(* IEC 61131-3 sources: verifaps-lib/geteta/examples/RTT_if (part 4) *)

        Pusher_states_t#Reset_interconnect_Slide1_Black:
             a_Pusher$_transit  := FALSE;
             a_Pusher$interconnect3  := FALSE;
             a_Pusher$Timer3$IN  := FALSE;
             a_Pusher$Timer3$PT  := USINT#0;
            IF  a_Pusher$Timer3$IN  THEN
                 a_Pusher$Timer3$Q  := ( a_Pusher$Timer3$ET  = USINT#0);
                IF ( a_Pusher$Timer3$ET  > USINT#0) THEN
                     a_Pusher$Timer3$ET  := ( a_Pusher$Timer3$ET  - USINT#1);
                ELSE
                     a_Pusher$Timer3$ET  := USINT#0;
                END_IF
            ELSE
                 a_Pusher$Timer3$Q  := FALSE;
                 a_Pusher$Timer3$ET  :=  a_Pusher$Timer3$PT ;
            END_IF
             a_Pusher$interconnect_Slide1_Black  := FALSE;
             a_Pusher$Timer_Slide1_Black$IN  := FALSE;
             a_Pusher$Timer_Slide1_Black$PT  := USINT#0;
            IF  a_Pusher$Timer_Slide1_Black$IN  THEN
                 a_Pusher$Timer_Slide1_Black$Q  := ( a_Pusher$Timer_Slide1_Black$ET  = USINT#0);
                IF ( a_Pusher$Timer_Slide1_Black$ET  > USINT#0) THEN
                     a_Pusher$Timer_Slide1_Black$ET  := ( a_Pusher$Timer_Slide1_Black$ET  - USINT#1);
                ELSE
                     a_Pusher$Timer_Slide1_Black$ET  := USINT#0;
                END_IF
            ELSE
                 a_Pusher$Timer_Slide1_Black$Q  := FALSE;
                 a_Pusher$Timer_Slide1_Black$ET  :=  a_Pusher$Timer_Slide1_Black$PT ;
            END_IF
             a_Pusher$Slide1_black  := ( a_Pusher$Slide1_black  - INT#1);
             a_Pusher$Priority_Var_Black  := ( a_Pusher$Priority_Var_Black  - INT#1);
            IF TRUE THEN
                 a_Pusher$_transit  := TRUE;
                 a_Pusher$_state  := Pusher_states_t#Interstep_2;
            END_IF

        Pusher_states_t#Reset_interconnect_Slide1_Metal:
             a_Pusher$_transit  := FALSE;
             a_Pusher$interconnect3  := FALSE;
             a_Pusher$Timer3$IN  := FALSE;
             a_Pusher$Timer3$PT  := USINT#0;
            IF  a_Pusher$Timer3$IN  THEN
                 a_Pusher$Timer3$Q  := ( a_Pusher$Timer3$ET  = USINT#0);
                IF ( a_Pusher$Timer3$ET  > USINT#0) THEN
                     a_Pusher$Timer3$ET  := ( a_Pusher$Timer3$ET  - USINT#1);
                ELSE
                     a_Pusher$Timer3$ET  := USINT#0;
                END_IF
            ELSE
                 a_Pusher$Timer3$Q  := FALSE;
                 a_Pusher$Timer3$ET  :=  a_Pusher$Timer3$PT ;
            END_IF
             a_Pusher$interconnect_Slide1_Metal  := FALSE;
             a_Pusher$Timer_Slide1_Metal$IN  := FALSE;
             a_Pusher$Timer_Slide1_Metal$PT  := USINT#0;
            IF  a_Pusher$Timer_Slide1_Metal$IN  THEN
                 a_Pusher$Timer_Slide1_Metal$Q  := ( a_Pusher$Timer_Slide1_Metal$ET  = USINT#0);
                IF ( a_Pusher$Timer_Slide1_Metal$ET  > USINT#0) THEN
                     a_Pusher$Timer_Slide1_Metal$ET  := ( a_Pusher$Timer_Slide1_Metal$ET  - USINT#1);
                ELSE
                     a_Pusher$Timer_Slide1_Metal$ET  := USINT#0;
                END_IF
            ELSE
                 a_Pusher$Timer_Slide1_Metal$Q  := FALSE;
                 a_Pusher$Timer_Slide1_Metal$ET  :=  a_Pusher$Timer_Slide1_Metal$PT ;
            END_IF
             a_Pusher$Slide1_metal  := ( a_Pusher$Slide1_metal  - INT#1);
             a_Pusher$Priority_Var_Metal  := ( a_Pusher$Priority_Var_Metal  - INT#1);
            IF TRUE THEN
                 a_Pusher$_transit  := TRUE;
                 a_Pusher$_state  := Pusher_states_t#Interstep_2;
            END_IF

        Pusher_states_t#Reset_interconnect_Slide1_White:
             a_Pusher$_transit  := FALSE;
             a_Pusher$interconnect3  := FALSE;
             a_Pusher$Timer3$IN  := FALSE;
             a_Pusher$Timer3$PT  := USINT#0;
            IF  a_Pusher$Timer3$IN  THEN
                 a_Pusher$Timer3$Q  := ( a_Pusher$Timer3$ET  = USINT#0);
                IF ( a_Pusher$Timer3$ET  > USINT#0) THEN
                     a_Pusher$Timer3$ET  := ( a_Pusher$Timer3$ET  - USINT#1);
                ELSE
                     a_Pusher$Timer3$ET  := USINT#0;
                END_IF
            ELSE
                 a_Pusher$Timer3$Q  := FALSE;
                 a_Pusher$Timer3$ET  :=  a_Pusher$Timer3$PT ;
            END_IF
             a_Pusher$interconnect_Slide1_White  := FALSE;
             a_Pusher$Timer_Slide1_White$IN  := FALSE;
             a_Pusher$Timer_Slide1_White$PT  := USINT#0;
            IF  a_Pusher$Timer_Slide1_White$IN  THEN
                 a_Pusher$Timer_Slide1_White$Q  := ( a_Pusher$Timer_Slide1_White$ET  = USINT#0);
                IF ( a_Pusher$Timer_Slide1_White$ET  > USINT#0) THEN
                     a_Pusher$Timer_Slide1_White$ET  := ( a_Pusher$Timer_Slide1_White$ET  - USINT#1);
                ELSE
                     a_Pusher$Timer_Slide1_White$ET  := USINT#0;
                END_IF
            ELSE
                 a_Pusher$Timer_Slide1_White$Q  := FALSE;
                 a_Pusher$Timer_Slide1_White$ET  :=  a_Pusher$Timer_Slide1_White$PT ;
            END_IF
             a_Pusher$Slide1_white  := ( a_Pusher$Slide1_white  - INT#1);
             a_Pusher$Priority_Var_White  := ( a_Pusher$Priority_Var_White  - INT#1);
            IF TRUE THEN
                 a_Pusher$_transit  := TRUE;
                 a_Pusher$_state  := Pusher_states_t#Interstep_2;
            END_IF

        Pusher_states_t#Reset_interconnect_Slide2_Black:
             a_Pusher$_transit  := FALSE;
             a_Pusher$interconnect3  := FALSE;
             a_Pusher$Timer3$IN  := FALSE;
             a_Pusher$Timer3$PT  := USINT#0;
            IF  a_Pusher$Timer3$IN  THEN
                 a_Pusher$Timer3$Q  := ( a_Pusher$Timer3$ET  = USINT#0);
                IF ( a_Pusher$Timer3$ET  > USINT#0) THEN
                     a_Pusher$Timer3$ET  := ( a_Pusher$Timer3$ET  - USINT#1);
                ELSE
                     a_Pusher$Timer3$ET  := USINT#0;
                END_IF
            ELSE
                 a_Pusher$Timer3$Q  := FALSE;
                 a_Pusher$Timer3$ET  :=  a_Pusher$Timer3$PT ;
            END_IF
             a_Pusher$interconnect_Slide2_Black  := FALSE;
             a_Pusher$Timer_Slide2_Black$IN  := FALSE;
             a_Pusher$Timer_Slide2_Black$PT  := USINT#0;
            IF  a_Pusher$Timer_Slide2_Black$IN  THEN
                 a_Pusher$Timer_Slide2_Black$Q  := ( a_Pusher$Timer_Slide2_Black$ET  = USINT#0);
                IF ( a_Pusher$Timer_Slide2_Black$ET  > USINT#0) THEN
                     a_Pusher$Timer_Slide2_Black$ET  := ( a_Pusher$Timer_Slide2_Black$ET  - USINT#1);
                ELSE
                     a_Pusher$Timer_Slide2_Black$ET  := USINT#0;
                END_IF
            ELSE
                 a_Pusher$Timer_Slide2_Black$Q  := FALSE;
                 a_Pusher$Timer_Slide2_Black$ET  :=  a_Pusher$Timer_Slide2_Black$PT ;
            END_IF
             a_Pusher$Slide2_black  := ( a_Pusher$Slide2_black  - INT#1);
             a_Pusher$Priority_Var_Black  := ( a_Pusher$Priority_Var_Black  - INT#1);
            IF TRUE THEN
                 a_Pusher$_transit  := TRUE;
                 a_Pusher$_state  := Pusher_states_t#Interstep_2;
            END_IF

        Pusher_states_t#Reset_interconnect_Slide2_Metal:
             a_Pusher$_transit  := FALSE;
             a_Pusher$interconnect3  := FALSE;
             a_Pusher$Timer3$IN  := FALSE;
             a_Pusher$Timer3$PT  := USINT#0;
            IF  a_Pusher$Timer3$IN  THEN
                 a_Pusher$Timer3$Q  := ( a_Pusher$Timer3$ET  = USINT#0);
                IF ( a_Pusher$Timer3$ET  > USINT#0) THEN
                     a_Pusher$Timer3$ET  := ( a_Pusher$Timer3$ET  - USINT#1);
                ELSE
                     a_Pusher$Timer3$ET  := USINT#0;
                END_IF
            ELSE
                 a_Pusher$Timer3$Q  := FALSE;
                 a_Pusher$Timer3$ET  :=  a_Pusher$Timer3$PT ;
            END_IF
             a_Pusher$interconnect_Slide2_Metal  := FALSE;
             a_Pusher$Timer_Slide2_Metal$IN  := FALSE;
             a_Pusher$Timer_Slide2_Metal$PT  := USINT#0;
            IF  a_Pusher$Timer_Slide2_Metal$IN  THEN
                 a_Pusher$Timer_Slide2_Metal$Q  := ( a_Pusher$Timer_Slide2_Metal$ET  = USINT#0);
                IF ( a_Pusher$Timer_Slide2_Metal$ET  > USINT#0) THEN
                     a_Pusher$Timer_Slide2_Metal$ET  := ( a_Pusher$Timer_Slide2_Metal$ET  - USINT#1);
                ELSE
                     a_Pusher$Timer_Slide2_Metal$ET  := USINT#0;
                END_IF
            ELSE
                 a_Pusher$Timer_Slide2_Metal$Q  := FALSE;
                 a_Pusher$Timer_Slide2_Metal$ET  :=  a_Pusher$Timer_Slide2_Metal$PT ;
            END_IF
             a_Pusher$Slide2_metal  := ( a_Pusher$Slide2_metal  - INT#1);
             a_Pusher$Priority_Var_Metal  := ( a_Pusher$Priority_Var_Metal  - INT#1);
            IF TRUE THEN
                 a_Pusher$_transit  := TRUE;
                 a_Pusher$_state  := Pusher_states_t#Interstep_2;
            END_IF

        Pusher_states_t#Reset_interconnect_Slide2_White:
             a_Pusher$_transit  := FALSE;
             a_Pusher$interconnect3  := FALSE;
             a_Pusher$Timer3$IN  := FALSE;
             a_Pusher$Timer3$PT  := USINT#0;
            IF  a_Pusher$Timer3$IN  THEN
                 a_Pusher$Timer3$Q  := ( a_Pusher$Timer3$ET  = USINT#0);
                IF ( a_Pusher$Timer3$ET  > USINT#0) THEN
                     a_Pusher$Timer3$ET  := ( a_Pusher$Timer3$ET  - USINT#1);
                ELSE
                     a_Pusher$Timer3$ET  := USINT#0;
                END_IF
            ELSE
                 a_Pusher$Timer3$Q  := FALSE;
                 a_Pusher$Timer3$ET  :=  a_Pusher$Timer3$PT ;
            END_IF
             a_Pusher$interconnect_Slide2_White  := FALSE;
             a_Pusher$Timer_Slide2_White$IN  := FALSE;
             a_Pusher$Timer_Slide2_White$PT  := USINT#0;
            IF  a_Pusher$Timer_Slide2_White$IN  THEN
                 a_Pusher$Timer_Slide2_White$Q  := ( a_Pusher$Timer_Slide2_White$ET  = USINT#0);
                IF ( a_Pusher$Timer_Slide2_White$ET  > USINT#0) THEN
                     a_Pusher$Timer_Slide2_White$ET  := ( a_Pusher$Timer_Slide2_White$ET  - USINT#1);
                ELSE
                     a_Pusher$Timer_Slide2_White$ET  := USINT#0;
                END_IF
            ELSE
                 a_Pusher$Timer_Slide2_White$Q  := FALSE;
                 a_Pusher$Timer_Slide2_White$ET  :=  a_Pusher$Timer_Slide2_White$PT ;
            END_IF
             a_Pusher$Slide2_white  := ( a_Pusher$Slide2_white  - INT#1);
             a_Pusher$Priority_Var_White  := ( a_Pusher$Priority_Var_White  - INT#1);
            IF TRUE THEN
                 a_Pusher$_transit  := TRUE;
                 a_Pusher$_state  := Pusher_states_t#Interstep_2;
            END_IF

        Pusher_states_t#Reset_interconnect_Slide3_Metal:
             a_Pusher$_transit  := FALSE;
             a_Pusher$interconnect3  := FALSE;
             a_Pusher$Timer3$IN  := FALSE;
             a_Pusher$Timer3$PT  := USINT#0;
            IF  a_Pusher$Timer3$IN  THEN
                 a_Pusher$Timer3$Q  := ( a_Pusher$Timer3$ET  = USINT#0);
                IF ( a_Pusher$Timer3$ET  > USINT#0) THEN
                     a_Pusher$Timer3$ET  := ( a_Pusher$Timer3$ET  - USINT#1);
                ELSE
                     a_Pusher$Timer3$ET  := USINT#0;
                END_IF
            ELSE
                 a_Pusher$Timer3$Q  := FALSE;
                 a_Pusher$Timer3$ET  :=  a_Pusher$Timer3$PT ;
            END_IF
             a_Pusher$Slide3_metal  := ( a_Pusher$Slide3_metal  - INT#1);
             a_Pusher$Priority_Var_Metal  := ( a_Pusher$Priority_Var_Metal  - INT#1);
            IF TRUE THEN
                 a_Pusher$_transit  := TRUE;
                 a_Pusher$_state  := Pusher_states_t#Interstep_2;
            END_IF

        Pusher_states_t#Reset_interconnect_Slide3_White:
             a_Pusher$_transit  := FALSE;
             a_Pusher$interconnect3  := FALSE;
             a_Pusher$Timer3$IN  := FALSE;
             a_Pusher$Timer3$PT  := USINT#0;
            IF  a_Pusher$Timer3$IN  THEN
                 a_Pusher$Timer3$Q  := ( a_Pusher$Timer3$ET  = USINT#0);
                IF ( a_Pusher$Timer3$ET  > USINT#0) THEN
                     a_Pusher$Timer3$ET  := ( a_Pusher$Timer3$ET  - USINT#1);
                ELSE
                     a_Pusher$Timer3$ET  := USINT#0;
                END_IF
            ELSE
                 a_Pusher$Timer3$Q  := FALSE;
                 a_Pusher$Timer3$ET  :=  a_Pusher$Timer3$PT ;
            END_IF
             a_Pusher$Slide3_white  := ( a_Pusher$Slide3_white  - INT#1);
             a_Pusher$Priority_Var_White  := ( a_Pusher$Priority_Var_White  - INT#1);
            IF TRUE THEN
                 a_Pusher$_transit  := TRUE;
                 a_Pusher$_state  := Pusher_states_t#Interstep_2;
            END_IF

        Pusher_states_t#Second_Slide_Timer_Black:
             a_Pusher$_transit  := FALSE;
            IF ( a_Pusher$SorterLightnesssensorCraneInterfaceInverse  = TRUE) THEN
                 a_Pusher$Timer_Slide2_Black$IN  :=  a_Pusher$SorterLightnesssensorCraneInterfaceInverse ;
                 a_Pusher$Timer_Slide2_Black$PT  :=  a_Pusher$Duration_Slide2_Black ;
                IF  a_Pusher$Timer_Slide2_Black$IN  THEN
                     a_Pusher$Timer_Slide2_Black$Q  := ( a_Pusher$Timer_Slide2_Black$ET  = USINT#0);
                    IF ( a_Pusher$Timer_Slide2_Black$ET  > USINT#0) THEN
                         a_Pusher$Timer_Slide2_Black$ET  := ( a_Pusher$Timer_Slide2_Black$ET  - USINT#1);
                    ELSE
                         a_Pusher$Timer_Slide2_Black$ET  := USINT#0;
                    END_IF
                ELSE
                     a_Pusher$Timer_Slide2_Black$Q  := FALSE;
                     a_Pusher$Timer_Slide2_Black$ET  :=  a_Pusher$Timer_Slide2_Black$PT ;
                END_IF
                 a_Pusher$interconnect_Slide2_Black  :=  a_Pusher$Timer_Slide2_Black$Q ;
            END_IF
            IF  a_Pusher$interconnect_Slide2_Black  THEN
                 a_Pusher$_transit  := TRUE;
                 a_Pusher$_state  := Pusher_states_t#PusherY2_Move_Out_Black;
            END_IF

        Pusher_states_t#Second_Slide_Timer_Metal:
             a_Pusher$_transit  := FALSE;
             a_Pusher$Timer_Slide2_Metal$IN  := TRUE;
             a_Pusher$Timer_Slide2_Metal$PT  :=  a_Pusher$Duration_Slide2_Metal ;
            IF  a_Pusher$Timer_Slide2_Metal$IN  THEN
                 a_Pusher$Timer_Slide2_Metal$Q  := ( a_Pusher$Timer_Slide2_Metal$ET  = USINT#0);
                IF ( a_Pusher$Timer_Slide2_Metal$ET  > USINT#0) THEN
                     a_Pusher$Timer_Slide2_Metal$ET  := ( a_Pusher$Timer_Slide2_Metal$ET  - USINT#1);
                ELSE
                     a_Pusher$Timer_Slide2_Metal$ET  := USINT#0;
                END_IF
            ELSE
                 a_Pusher$Timer_Slide2_Metal$Q  := FALSE;
                 a_Pusher$Timer_Slide2_Metal$ET  :=  a_Pusher$Timer_Slide2_Metal$PT ;
            END_IF
             a_Pusher$interconnect_Slide2_Metal  :=  a_Pusher$Timer_Slide2_Metal$Q ;
            IF  a_Pusher$interconnect_Slide2_Metal  THEN
                 a_Pusher$_transit  := TRUE;
                 a_Pusher$_state  := Pusher_states_t#PusherY2_Move_Out_Metal;
            END_IF

        Pusher_states_t#Second_Slide_Timer_White:
             a_Pusher$_transit  := FALSE;
             a_Pusher$Timer_Slide2_White$IN  := TRUE;
             a_Pusher$Timer_Slide2_White$PT  :=  a_Pusher$Duration_Slide2_White ;
            IF  a_Pusher$Timer_Slide2_White$IN  THEN
                 a_Pusher$Timer_Slide2_White$Q  := ( a_Pusher$Timer_Slide2_White$ET  = USINT#0);
                IF ( a_Pusher$Timer_Slide2_White$ET  > USINT#0) THEN
                     a_Pusher$Timer_Slide2_White$ET  := ( a_Pusher$Timer_Slide2_White$ET  - USINT#1);
                ELSE
                     a_Pusher$Timer_Slide2_White$ET  := USINT#0;
                END_IF
            ELSE
                 a_Pusher$Timer_Slide2_White$Q  := FALSE;
                 a_Pusher$Timer_Slide2_White$ET  :=  a_Pusher$Timer_Slide2_White$PT ;
            END_IF
             a_Pusher$interconnect_Slide2_White  :=  a_Pusher$Timer_Slide2_White$Q ;
            IF  a_Pusher$interconnect_Slide2_White  THEN
                 a_Pusher$_transit  := TRUE;
                 a_Pusher$_state  := Pusher_states_t#PusherY2_Move_Out_White;
            END_IF

        Pusher_states_t#Second_Slide_black_workpieces:
             a_Pusher$_transit  := FALSE;
            IF TRUE THEN
                 a_Pusher$_transit  := TRUE;
                 a_Pusher$_state  := Pusher_states_t#Second_Slide_Timer_Black;
            END_IF

        Pusher_states_t#Second_Slide_metal_workpieces:
             a_Pusher$_transit  := FALSE;
            IF ( a_Pusher$SorterLightnessSensorPusher2  AND  a_Pusher$SorterCapacitiveSensorPusher2 ) THEN
                 a_Pusher$_transit  := TRUE;
                 a_Pusher$_state  := Pusher_states_t#Second_Test_For_Metal;
            END_IF

        Pusher_states_t#Second_Slide_white_workpieces:
             a_Pusher$_transit  := FALSE;
            IF ( a_Pusher$SorterLightnessSensorPusher2  AND NOT  a_Pusher$SorterCapacitiveSensorPusher2 ) THEN
                 a_Pusher$_transit  := TRUE;
                 a_Pusher$_state  := Pusher_states_t#Second_Test_For_White;
            END_IF

        Pusher_states_t#Second_Test_For_Metal:
             a_Pusher$_transit  := FALSE;
            IF TRUE THEN
                 a_Pusher$_transit  := TRUE;
                 a_Pusher$_state  := Pusher_states_t#Second_Slide_Timer_Metal;
            END_IF

        Pusher_states_t#Second_Test_For_White:
             a_Pusher$_transit  := FALSE;
            IF TRUE THEN
                 a_Pusher$_transit  := TRUE;
                 a_Pusher$_state  := Pusher_states_t#Second_Slide_Timer_White;
            END_IF

        Pusher_states_t#Third_Slide_black_workpieces:
             a_Pusher$_transit  := FALSE;
            IF (NOT  a_Pusher$SorterLightnessSensorPusher2  AND NOT  a_Pusher$SorterCapacitiveSensorPusher2 ) THEN
                 a_Pusher$_transit  := TRUE;
                 a_Pusher$_state  := Pusher_states_t#Wait_Black;
            END_IF

        Pusher_states_t#Third_Slide_metal_workpieces:
             a_Pusher$_transit  := FALSE;
            IF ( a_Pusher$SorterLightnessSensorPusher2  AND  a_Pusher$SorterCapacitiveSensorPusher2 ) THEN
                 a_Pusher$_transit  := TRUE;
                 a_Pusher$_state  := Pusher_states_t#Wait_Metal;
            END_IF

        Pusher_states_t#Third_Slide_white_workpieces:
             a_Pusher$_transit  := FALSE;
            IF ( a_Pusher$SorterLightnessSensorPusher2  AND NOT  a_Pusher$SorterCapacitiveSensorPusher2 ) THEN
                 a_Pusher$_transit  := TRUE;
                 a_Pusher$_state  := Pusher_states_t#Wait_White;
            END_IF

        Pusher_states_t#Wait_Black:
             a_Pusher$_transit  := FALSE;
            IF ((NOT  a_Pusher$SorterLightnessSensorPusher2  AND NOT  a_Pusher$SorterCapacitiveSensorPusher2 ) = TRUE) THEN
                 a_Pusher$Timer2$IN  := (NOT  a_Pusher$SorterLightnessSensorPusher2  AND NOT  a_Pusher$SorterCapacitiveSensorPusher2 );
                 a_Pusher$Timer2$PT  :=  a_Pusher$Duration2 ;
                IF  a_Pusher$Timer2$IN  THEN
                     a_Pusher$Timer2$Q  := ( a_Pusher$Timer2$ET  = USINT#0);
                    IF ( a_Pusher$Timer2$ET  > USINT#0) THEN
                         a_Pusher$Timer2$ET  := ( a_Pusher$Timer2$ET  - USINT#1);
                    ELSE
                         a_Pusher$Timer2$ET  := USINT#0;
                    END_IF
                ELSE
                     a_Pusher$Timer2$Q  := FALSE;
                     a_Pusher$Timer2$ET  :=  a_Pusher$Timer2$PT ;
                END_IF
                 a_Pusher$interconnect2  :=  a_Pusher$Timer2$Q ;
            END_IF
            IF  a_Pusher$interconnect2  THEN
                 a_Pusher$_transit  := TRUE;
                 a_Pusher$_state  := Pusher_states_t#Reset_interconnect3;
            END_IF

        Pusher_states_t#Wait_Metal:
             a_Pusher$_transit  := FALSE;
             a_Pusher$Timer3$IN  := TRUE;
             a_Pusher$Timer3$PT  :=  a_Pusher$Duration3 ;
            IF  a_Pusher$Timer3$IN  THEN
                 a_Pusher$Timer3$Q  := ( a_Pusher$Timer3$ET  = USINT#0);
                IF ( a_Pusher$Timer3$ET  > USINT#0) THEN
                     a_Pusher$Timer3$ET  := ( a_Pusher$Timer3$ET  - USINT#1);
                ELSE
                     a_Pusher$Timer3$ET  := USINT#0;
                END_IF
            ELSE
                 a_Pusher$Timer3$Q  := FALSE;
                 a_Pusher$Timer3$ET  :=  a_Pusher$Timer3$PT ;
            END_IF
             a_Pusher$interconnect3  :=  a_Pusher$Timer3$Q ;
            IF  a_Pusher$interconnect3  THEN
                 a_Pusher$_transit  := TRUE;
                 a_Pusher$_state  := Pusher_states_t#Reset_interconnect_Slide3_Metal;
            END_IF

        Pusher_states_t#Wait_White:
             a_Pusher$_transit  := FALSE;
             a_Pusher$Timer3$IN  := TRUE;
             a_Pusher$Timer3$PT  :=  a_Pusher$Duration3 ;
            IF  a_Pusher$Timer3$IN  THEN
                 a_Pusher$Timer3$Q  := ( a_Pusher$Timer3$ET  = USINT#0);
                IF ( a_Pusher$Timer3$ET  > USINT#0) THEN
                     a_Pusher$Timer3$ET  := ( a_Pusher$Timer3$ET  - USINT#1);
                ELSE
                     a_Pusher$Timer3$ET  := USINT#0;
                END_IF
            ELSE
                 a_Pusher$Timer3$Q  := FALSE;
                 a_Pusher$Timer3$ET  :=  a_Pusher$Timer3$PT ;
            END_IF
             a_Pusher$interconnect3  :=  a_Pusher$Timer3$Q ;
            IF  a_Pusher$interconnect3  THEN
                 a_Pusher$_transit  := TRUE;
                 a_Pusher$_state  := Pusher_states_t#Reset_interconnect_Slide3_White;
            END_IF

        Pusher_states_t#Wait_Y1_Black:
             a_Pusher$_transit  := FALSE;
            IF ( a_Pusher$PusherY1  = TRUE) THEN
                 a_Pusher$Timer3$IN  :=  a_Pusher$PusherY1 ;
                 a_Pusher$Timer3$PT  :=  a_Pusher$Duration3 ;
                IF  a_Pusher$Timer3$IN  THEN
                     a_Pusher$Timer3$Q  := ( a_Pusher$Timer3$ET  = USINT#0);
                    IF ( a_Pusher$Timer3$ET  > USINT#0) THEN
                         a_Pusher$Timer3$ET  := ( a_Pusher$Timer3$ET  - USINT#1);
                    ELSE
                         a_Pusher$Timer3$ET  := USINT#0;
                    END_IF
                ELSE
                     a_Pusher$Timer3$Q  := FALSE;
                     a_Pusher$Timer3$ET  :=  a_Pusher$Timer3$PT ;
                END_IF
                 a_Pusher$interconnect3  :=  a_Pusher$Timer3$Q ;
            END_IF
            IF  a_Pusher$interconnect3  THEN
                 a_Pusher$_transit  := TRUE;
                 a_Pusher$_state  := Pusher_states_t#PusherY1_Move_In_Black;
            END_IF

        Pusher_states_t#Wait_Y1_Metal:
             a_Pusher$_transit  := FALSE;
            IF ( a_Pusher$PusherY1  = TRUE) THEN
                 a_Pusher$Timer3$IN  :=  a_Pusher$PusherY1 ;
                 a_Pusher$Timer3$PT  :=  a_Pusher$Duration3 ;
                IF  a_Pusher$Timer3$IN  THEN
                     a_Pusher$Timer3$Q  := ( a_Pusher$Timer3$ET  = USINT#0);
                    IF ( a_Pusher$Timer3$ET  > USINT#0) THEN
                         a_Pusher$Timer3$ET  := ( a_Pusher$Timer3$ET  - USINT#1);
                    ELSE
                         a_Pusher$Timer3$ET  := USINT#0;
                    END_IF
                ELSE
                     a_Pusher$Timer3$Q  := FALSE;
                     a_Pusher$Timer3$ET  :=  a_Pusher$Timer3$PT ;
                END_IF
                 a_Pusher$interconnect3  :=  a_Pusher$Timer3$Q ;
            END_IF
            IF  a_Pusher$interconnect3  THEN
                 a_Pusher$_transit  := TRUE;
                 a_Pusher$_state  := Pusher_states_t#PusherY1_Move_In_Metal;
            END_IF

        Pusher_states_t#Wait_Y1_White:
             a_Pusher$_transit  := FALSE;
            IF ( a_Pusher$PusherY1  = TRUE) THEN
                 a_Pusher$Timer3$IN  :=  a_Pusher$PusherY1 ;
                 a_Pusher$Timer3$PT  :=  a_Pusher$Duration3 ;
                IF  a_Pusher$Timer3$IN  THEN
                     a_Pusher$Timer3$Q  := ( a_Pusher$Timer3$ET  = USINT#0);
                    IF ( a_Pusher$Timer3$ET  > USINT#0) THEN
                         a_Pusher$Timer3$ET  := ( a_Pusher$Timer3$ET  - USINT#1);
                    ELSE
                         a_Pusher$Timer3$ET  := USINT#0;
                    END_IF
                ELSE
                     a_Pusher$Timer3$Q  := FALSE;
                     a_Pusher$Timer3$ET  :=  a_Pusher$Timer3$PT ;
                END_IF
                 a_Pusher$interconnect3  :=  a_Pusher$Timer3$Q ;
            END_IF
            IF  a_Pusher$interconnect3  THEN
                 a_Pusher$_transit  := TRUE;
                 a_Pusher$_state  := Pusher_states_t#PusherY1_Move_In_White;
            END_IF

        Pusher_states_t#Wait_Y2_Black:
             a_Pusher$_transit  := FALSE;
            IF ( a_Pusher$PusherY2  = TRUE) THEN
                 a_Pusher$Timer3$IN  :=  a_Pusher$PusherY2 ;
                 a_Pusher$Timer3$PT  :=  a_Pusher$Duration3 ;
                IF  a_Pusher$Timer3$IN  THEN
                     a_Pusher$Timer3$Q  := ( a_Pusher$Timer3$ET  = USINT#0);
                    IF ( a_Pusher$Timer3$ET  > USINT#0) THEN
                         a_Pusher$Timer3$ET  := ( a_Pusher$Timer3$ET  - USINT#1);
                    ELSE
                         a_Pusher$Timer3$ET  := USINT#0;
                    END_IF
                ELSE
                     a_Pusher$Timer3$Q  := FALSE;
                     a_Pusher$Timer3$ET  :=  a_Pusher$Timer3$PT ;
                END_IF
                 a_Pusher$interconnect3  :=  a_Pusher$Timer3$Q ;
            END_IF
            IF  a_Pusher$interconnect3  THEN
                 a_Pusher$_transit  := TRUE;
                 a_Pusher$_state  := Pusher_states_t#PusherY2_Move_In_Black;
            END_IF

        Pusher_states_t#Wait_Y2_Metal:
             a_Pusher$_transit  := FALSE;
            IF ( a_Pusher$PusherY2  = TRUE) THEN
                 a_Pusher$Timer3$IN  :=  a_Pusher$PusherY2 ;
                 a_Pusher$Timer3$PT  :=  a_Pusher$Duration3 ;
                IF  a_Pusher$Timer3$IN  THEN
                     a_Pusher$Timer3$Q  := ( a_Pusher$Timer3$ET  = USINT#0);
                    IF ( a_Pusher$Timer3$ET  > USINT#0) THEN
                         a_Pusher$Timer3$ET  := ( a_Pusher$Timer3$ET  - USINT#1);
                    ELSE
                         a_Pusher$Timer3$ET  := USINT#0;
                    END_IF
                ELSE
                     a_Pusher$Timer3$Q  := FALSE;
                     a_Pusher$Timer3$ET  :=  a_Pusher$Timer3$PT ;
                END_IF
                 a_Pusher$interconnect3  :=  a_Pusher$Timer3$Q ;
            END_IF
            IF  a_Pusher$interconnect3  THEN
                 a_Pusher$_transit  := TRUE;
                 a_Pusher$_state  := Pusher_states_t#PusherY2_Move_In_Metal;
            END_IF

        Pusher_states_t#Wait_Y2_White:
             a_Pusher$_transit  := FALSE;
            IF ( a_Pusher$PusherY2  = TRUE) THEN
                 a_Pusher$Timer3$IN  :=  a_Pusher$PusherY2 ;
                 a_Pusher$Timer3$PT  :=  a_Pusher$Duration3 ;
                IF  a_Pusher$Timer3$IN  THEN
                     a_Pusher$Timer3$Q  := ( a_Pusher$Timer3$ET  = USINT#0);
                    IF ( a_Pusher$Timer3$ET  > USINT#0) THEN
                         a_Pusher$Timer3$ET  := ( a_Pusher$Timer3$ET  - USINT#1);
                    ELSE
                         a_Pusher$Timer3$ET  := USINT#0;
                    END_IF
                ELSE
                     a_Pusher$Timer3$Q  := FALSE;
                     a_Pusher$Timer3$ET  :=  a_Pusher$Timer3$PT ;
                END_IF
                 a_Pusher$interconnect3  :=  a_Pusher$Timer3$Q ;
            END_IF
            IF  a_Pusher$interconnect3  THEN
                 a_Pusher$_transit  := TRUE;
                 a_Pusher$_state  := Pusher_states_t#PusherY2_Move_In_White;
            END_IF

            END_CASE
    IF (( a_Actuator_SorterGreenLampConveyor  AND  a_Actuator_MagazinGreenLamp ) AND  a_Actuator_StampGreenLamp ) THEN
        IF ((( a_Stamp$StartCommandStamp  AND  a_Crane$StartCommandCrane ) AND  a_Conveyor$StartCommandConveyor ) AND  a_Mag$StartCommandMagazin ) THEN
             a_Crane$StartVar  := TRUE;
             a_Conveyor$StartVar  := TRUE;
             a_Mag$StartVar  := TRUE;
             a_Pusher$StartVar  := TRUE;
             a_Stamp$StartVar  := TRUE;
             a_DIAGNOSIS_ACTIVE  := TRUE;
        END_IF
    END_IF
     a_Crane$SFCReset  := FALSE;
     a_Conveyor$SFCReset  := FALSE;
     a_Mag$SFCReset  := FALSE;
     a_Pusher$SFCReset  := FALSE;
     a_Stamp$SFCReset  := FALSE;

     a_Crane$AnalogCranePressure  :=  a_PARAMETER_CRANE_PRESSURE_METALLIC ;

ELSEIF ((NOT  a_Sensor_SorterEmergencyStop  OR NOT  a_Sensor_StampEmergencyStop ) OR NOT  a_Sensor_MagazinEmergencyStop ) THEN
     a_Actuator_MagazinSlider  := FALSE;
     a_Actuator_CraneLower  := FALSE;
     a_Actuator_MagazinVacuumOn  := FALSE;
     a_Actuator_MagazinVacuumOff  := TRUE;
     a_Actuator_MagazinGreenLamp  := FALSE;
     a_Actuator_CraneTurnCounterclockwise  := FALSE;
     a_Actuator_CraneTurnClockwise  := FALSE;
     a_Actuator_SorterConveyorTowardsStacker  := FALSE;
     a_Actuator_SorterConveyorTowardsCrane  := FALSE;
     a_Actuator_SorterGreenLampConveyor  := FALSE;
     a_Actuator_PusherY1  := FALSE;
     a_Actuator_PusherY2  := FALSE;
     a_Actuator_StampSliderMovedOut  := TRUE;
     a_Actuator_StampSliderMovedIn  := FALSE;
     a_Actuator_StampGreenLamp  := FALSE;
     a_Actuator_StampPusher  := FALSE;
     a_Actuator_AnalogCranePressure  := INT#0;
     a_Crane$SFCReset  := TRUE;
     a_Conveyor$SFCReset  := TRUE;
     a_Mag$SFCReset  := TRUE;
     a_Pusher$SFCReset  := TRUE;
     a_Stamp$SFCReset  := TRUE;
     a_Crane$StartVar  := FALSE;
     a_Conveyor$StartVar  := FALSE;
     a_Mag$StartVar  := FALSE;
     a_Pusher$StartVar  := FALSE;
     a_Stamp$StartVar  := FALSE;
END_IF

//--------------------------------------------------------------------------------

 b_Mag$SliderNotMovedOut  :=  b_Sensor_SliderNotMovedOut ;
 b_Mag$SliderMovedOut  :=  b_Sensor_SliderMovedOut ;
 b_Mag$CraneOnMagazin  :=  b_Sensor_CraneOnMagazin ;
 b_Mag$CraneDown  :=  b_Sensor_CraneDown ;
 b_Mag$CraneUp  :=  b_Sensor_CraneUp ;
 b_Mag$CraneOnConveyor  :=  b_Sensor_CraneOnConveyor ;
 b_Mag$WorkpieceReady  :=  b_Sensor_WorkpieceReady ;
 b_Mag$AnalogCranePosition  :=  b_Sensor_AnalogCranePosition ;
 b_Mag$StartButtonMagazin  :=  b_Sensor_StartButtonMagazin ;
 b_Actuator_MagazinSlider  :=  b_Mag$MagazinSlider ;
 b_Actuator_MagazinGreenLamp  :=  b_Mag$MagazinGreenLamp ;
 b_Crane$CraneUp  :=  b_Sensor_CraneUp ;
 b_Crane$CraneDown  :=  b_Sensor_CraneDown ;
 b_Crane$CraneSucked  :=  b_Sensor_CraneSucked ;
 b_Crane$MagazinCapacitiveSensor  :=  b_Sensor_MagazinCapacitiveSensor ;
 b_Crane$SliderMovedOut  :=  b_Sensor_SliderMovedOut ;
 b_Crane$WorkpieceReady  :=  b_Sensor_WorkpieceReady ;
 b_Crane$MagazinOpticalSensor  :=  b_Sensor_MagazinOpticalSensor ;
 b_Crane$StampSliderFilled  :=  b_Sensor_StampSliderFilled ;
 b_Crane$StampSliderSensorMovedOut  :=  b_Sensor_StampSliderSensorMovedOut ;
 b_Crane$StampLowered  :=  b_Sensor_StampLowered ;
 b_Crane$AnalogCranePosition  :=  b_Sensor_AnalogCranePosition ;
 b_Crane$StartButtonMagazin  :=  b_Sensor_StartButtonMagazin ;

//Diagnosis
// old:  b_Actuator_AnalogCranePressure
// new:  b_Crane$AnalogCranePressure ;
 b_Actuator_CraneTurnCounterclockwise  :=  b_Crane$CraneTurnCounterclockwise ;
 b_Actuator_CraneTurnClockwise  :=  b_Crane$CraneTurnClockwise ;

IF  b_DIAGNOSIS_ACTIVE  THEN
        IF  b_Sensor_CraneSucked  AND ( b_Crane$AnalogCranePressure  <= 0 OR  b_Crane$AnalogCranePressure  > 10000) THEN
                 b_Actuator_CraneTurnCounterclockwise  := FALSE;
                 b_Actuator_CraneTurnClockwise  := FALSE;
        END_IF
END_IF

//End of Diagnosis

 b_Actuator_CraneLower  :=  b_Crane$CraneLower ;
 b_Actuator_MagazinVacuumOff  :=  b_Crane$MagazinVacuumOff ;
 b_Actuator_MagazinVacuumOn  :=  b_Crane$MagazinVacuumOn ;
 b_Actuator_AnalogCranePressure  :=  b_Crane$AnalogCranePressure ;
 b_Stamp$StampSliderSensorMovedOut  :=  b_Sensor_StampSliderSensorMovedOut ;
 b_Stamp$StampSliderSensorMovedIn  :=  b_Sensor_StampSliderSensorMovedIn ;
 b_Stamp$StampSliderFilled  :=  b_Sensor_StampSliderFilled ;
 b_Stamp$StampUp  :=  b_Sensor_StampUp ;
 b_Stamp$StampLowered  :=  b_Sensor_StampLowered ;
 b_Stamp$CraneDown  :=  b_Sensor_CraneDown ;
 b_Stamp$CraneUp  :=  b_Sensor_CraneUp ;
 b_Stamp$CraneSucked  :=  b_Sensor_CraneSucked ;
 b_Stamp$CranePositionStamp  :=  b_Sensor_CranePositionStamp ;
 b_Stamp$CraneOnConveyor  :=  b_Sensor_CraneOnConveyor ;
 b_Stamp$AnalogCranePosition  :=  b_Sensor_AnalogCranePosition ;
 b_Stamp$StampStartButton  :=  b_Sensor_StampStartButton ;
 b_Actuator_StampSliderMovedOut  :=  b_Stamp$StampSliderMovedOut ;
 b_Actuator_StampSliderMovedIn  :=  b_Stamp$StampSliderMovedIn ;
 b_Actuator_StampWhiteLamp  :=  b_Stamp$StampWhiteLamp ;
 b_Actuator_StampPusher  :=  b_Stamp$StampPusher ;
 b_Actuator_StampGreenLamp  :=  b_Stamp$StampGreenLamp ;
 b_Conveyor$SorterStartButton  :=  b_Sensor_SorterStartButton ;
 b_Conveyor$SorterSwitchManuellAutomatic  :=  b_Sensor_SorterSwitchManuellAutomatic ;
 b_Conveyor$SorterLightbarrierCraneInterface  :=  b_Sensor_SorterLightbarrierCraneInterface ;
 b_Actuator_SorterConveyorTowardsStacker  :=  b_Conveyor$SorterConveyorTowardsStacker ;
 b_Actuator_SorterConveyorTowardsCrane  :=  b_Conveyor$SorterConveyorTowardsCrane ;
 b_Actuator_SorterGreenLampConveyor  :=  b_Conveyor$SorterGreenLampConveyor ;
 b_Actuator_SorterWhiteLampConveyor  :=  b_Conveyor$SorterWhiteLampConveyor ;
 b_Pusher$SorterLightnesssensorCraneInterfaceInverse  :=  b_Sensor_SorterLightnesssensorCraneInterfaceInverse ;
 b_Pusher$SorterLightbarrierCraneInterface  :=  b_Sensor_SorterLightbarrierCraneInterface ;
 b_Pusher$SorterCapacitiveSensorPusher1  :=  b_Sensor_SorterCapacitiveSensorPusher1 ;
 b_Pusher$SorterLightnessSensorPusher1  :=  b_Sensor_SorterLightnessSensorPusher1 ;
 b_Pusher$SorterCapacitiveSensorPusher2  :=  b_Sensor_SorterCapacitiveSensorPusher2 ;
 b_Pusher$SorterLightnessSensorPusher2  :=  b_Sensor_SorterLightnessSensorPusher2 ;
 b_Pusher$SorterLightnessSensorPusher3  :=  b_Sensor_SorterLightnessSensorPusher3 ;
 b_Pusher$SorterPusher1MovedOut  :=  b_Sensor_SorterPusher1MovedOut ;
 b_Pusher$SorterPusher1MovedIn  :=  b_Sensor_SorterPusher1MovedIn ;
 b_Pusher$SorterPusher2MovedOut  :=  b_Sensor_SorterPusher2MovedOut ;
 b_Pusher$SorterPusher2MovedIn  :=  b_Sensor_SorterPusher2MovedIn ;
 b_Pusher$SorterStartButton  :=  b_Sensor_SorterStartButton ;
 b_Actuator_PusherY1  :=  b_Pusher$PusherY1 ;
 b_Actuator_PusherY2  :=  b_Pusher$PusherY2 ;

IF (( b_Sensor_SorterEmergencyStop  AND  b_Sensor_StampEmergencyStop ) AND  b_Sensor_MagazinEmergencyStop ) THEN
    CASE  b_Mag$_state  OF
        Magazin_states_t#Green_Lamp:
             b_Mag$_transit  := FALSE;
             b_Mag$MagazinGreenLamp  := TRUE;
             b_Mag$interconnectMagazinStartCommand  := FALSE;
            IF TRUE THEN
                 b_Mag$_transit  := TRUE;
                 b_Mag$_state  := Magazin_states_t#Magazin_Init;
            END_IF

        Magazin_states_t#Init:
             b_Mag$_transit  := FALSE;
            IF TRUE THEN
                 b_Mag$_transit  := TRUE;
                 b_Mag$_state  := Magazin_states_t#Start_Magazin;
            END_IF

        Magazin_states_t#Interstep:
             b_Mag$_transit  := FALSE;
             b_Mag$StartCommandMagazin  := TRUE;
            IF  b_Mag$StartVar  THEN
                 b_Mag$_transit  := TRUE;
                 b_Mag$_state  := Magazin_states_t#convey;
            END_IF

        Magazin_states_t#Magazin_Init:
             b_Mag$_transit  := FALSE;
             b_Mag$MagazinSlider  := TRUE;
            IF TRUE THEN
                 b_Mag$_transit  := TRUE;
                 b_Mag$_state  := Magazin_states_t#Magazin_Init_2;
            END_IF

        Magazin_states_t#Magazin_Init_2:
             b_Mag$_transit  := FALSE;
             b_Mag$MagazinSlider  := FALSE;
            IF TRUE THEN
                 b_Mag$_transit  := TRUE;
                 b_Mag$_state  := Magazin_states_t#Interstep;
            END_IF

        Magazin_states_t#Slider_Move_Back:
             b_Mag$_transit  := FALSE;
            IF (( b_Mag$SliderMovedOut  = TRUE) AND ( b_Mag$SliderNotMovedOut  = FALSE)) THEN
                 b_Mag$MagazinSlider  := FALSE;
            END_IF
            IF  b_Mag$CraneUp  THEN
                 b_Mag$_transit  := TRUE;
                 b_Mag$_state  := Magazin_states_t#Step1;
            END_IF

        Magazin_states_t#Start_Magazin:
             b_Mag$_transit  := FALSE;
             b_Mag$MagazinSlider  := FALSE;
             b_Mag$MagazinGreenLamp  := FALSE;
             b_Mag$StartVar  := FALSE;
             b_Mag$StartCommandMagazin  := FALSE;
            IF ( b_Mag$StartButtonMagazin  = TRUE) THEN
                 b_Mag$interconnectMagazinStartCommand  := TRUE;
            END_IF
            IF  b_Mag$interconnectMagazinStartCommand  THEN
                 b_Mag$_transit  := TRUE;
                 b_Mag$_state  := Magazin_states_t#Green_Lamp;
            END_IF

        Magazin_states_t#Step0:
             b_Mag$_transit  := FALSE;
            IF  b_Mag$CraneDown  THEN
                 b_Mag$_transit  := TRUE;
                 b_Mag$_state  := Magazin_states_t#Slider_Move_Back;
            END_IF

        Magazin_states_t#Step1:
             b_Mag$_transit  := FALSE;
            IF (( b_Mag$AnalogCranePosition  > INT#16160) AND ( b_Mag$AnalogCranePosition  < INT#16260)) THEN
                 b_Mag$_transit  := TRUE;
                 b_Mag$_state  := Magazin_states_t#Interstep;
            END_IF

        Magazin_states_t#convey:
             b_Mag$_transit  := FALSE;
            IF  b_Mag$SliderNotMovedOut  THEN
                 b_Mag$MagazinSlider  := TRUE;
            END_IF
            IF (( b_Mag$AnalogCranePosition  > INT#24290) AND ( b_Mag$AnalogCranePosition  < INT#24390)) THEN
                 b_Mag$_transit  := TRUE;
                 b_Mag$_state  := Magazin_states_t#Step0;
            END_IF

            END_CASE
    CASE  b_Crane$_state  OF
        Crane_states_t#Crane_Go_Up:
             b_Crane$_transit  := FALSE;
             b_Crane$CraneLower  := FALSE;
            IF  b_Crane$CraneUp  THEN
                 b_Crane$_transit  := TRUE;
                 b_Crane$_state  := Crane_states_t#Step3;
            END_IF

        Crane_states_t#Crane_Go_Up_White:
             b_Crane$_transit  := FALSE;
             b_Crane$CraneLower  := FALSE;
            IF  b_Crane$CraneUp  THEN
                 b_Crane$_transit  := TRUE;
                 b_Crane$_state  := Crane_states_t#Step3;
            END_IF

        Crane_states_t#Crane_Init:
             b_Crane$_transit  := FALSE;
             b_Crane$CraneLower  := TRUE;
             b_Crane$interconnectCraneStartCommand  := FALSE;
             b_Crane$AnalogCranePressure  :=  b_PARAMETER_CRANE_PRESSURE_METALLIC ;
            IF  b_Crane$CraneDown  THEN
                 b_Crane$_transit  := TRUE;
                 b_Crane$_state  := Crane_states_t#Crane_Init_2;
            END_IF

        Crane_states_t#Crane_Init_2:
             b_Crane$_transit  := FALSE;
             b_Crane$CraneLower  := FALSE;
            IF  b_Crane$CraneUp  THEN
                 b_Crane$_transit  := TRUE;
                 b_Crane$_state  := Crane_states_t#Interstep;
            END_IF

        Crane_states_t#Crane_Lift_At_Stamp:
             b_Crane$_transit  := FALSE;
             b_Crane$CraneLower  := FALSE;
            IF  b_Crane$CraneUp  THEN
                 b_Crane$_transit  := TRUE;
                 b_Crane$_state  := Crane_states_t#Crane_Turn_Left_From_Stamp;
            END_IF

        Crane_states_t#Crane_Lift_At_Stamp2:
             b_Crane$_transit  := FALSE;
             b_Crane$CraneLower  := FALSE;
             b_Crane$AnalogCranePressure  := INT#0;
            IF  b_Crane$CraneUp  THEN
                 b_Crane$_transit  := TRUE;
                 b_Crane$_state  := Crane_states_t#Crane_Turn_Right_From_Stamp;
            END_IF

        Crane_states_t#Crane_Lift_Conveyor:
             b_Crane$_transit  := FALSE;
             b_Crane$CraneLower  := FALSE;
            IF TRUE THEN
                 b_Crane$_transit  := TRUE;
                 b_Crane$_state  := Crane_states_t#Interstep;
            END_IF

        Crane_states_t#Crane_Lift_Conveyor2:
             b_Crane$_transit  := FALSE;
             b_Crane$CraneLower  := FALSE;
            IF TRUE THEN
                 b_Crane$_transit  := TRUE;
                 b_Crane$_state  := Crane_states_t#Interstep;
            END_IF

        Crane_states_t#Crane_Lift_Conveyor_Black:
             b_Crane$_transit  := FALSE;
             b_Crane$CraneLower  := FALSE;
            IF  b_Crane$CraneUp  THEN
                 b_Crane$_transit  := TRUE;
                 b_Crane$_state  := Crane_states_t#Crane_Turn_Left_Back_To_Stamp;
            END_IF

        Crane_states_t#Crane_Lift_Magazin:
             b_Crane$_transit  := FALSE;
             b_Crane$CraneLower  := FALSE;
            IF  b_Crane$CraneUp  THEN
                 b_Crane$_transit  := TRUE;
                 b_Crane$_state  := Crane_states_t#Crane_Turn_Left_NOT_Metallic;
            END_IF

        Crane_states_t#Crane_Lift_Magazin_Metallic:
             b_Crane$_transit  := FALSE;
             b_Crane$CraneLower  := FALSE;
            IF  b_Crane$CraneUp  THEN
                 b_Crane$_transit  := TRUE;
                 b_Crane$_state  := Crane_states_t#Crane_Turn_Left_Metallic;
            END_IF

        Crane_states_t#Crane_Lift_Magazin_White:
             b_Crane$_transit  := FALSE;
             b_Crane$CraneLower  := FALSE;
            IF  b_Crane$CraneUp  THEN
                 b_Crane$_transit  := TRUE;
                 b_Crane$_state  := Crane_states_t#Crane_Turn_Left_White;
            END_IF

        Crane_states_t#Crane_Lift_NOT_Metallic_Black:
             b_Crane$_transit  := FALSE;
             b_Crane$CraneLower  := FALSE;
            IF  b_Crane$CraneUp  THEN
                 b_Crane$_transit  := TRUE;
                 b_Crane$_state  := Crane_states_t#Crane_Turn_Left_NOT_Metallic_Black;
            END_IF

        Crane_states_t#Crane_Lower:
             b_Crane$_transit  := FALSE;
             b_Crane$MagazinVacuumOn  := TRUE;
             b_Crane$MagazinVacuumOff  := FALSE;
             b_Crane$CraneLower  := TRUE;
             b_Crane$AnalogCranePressure  := INT#0;
            IF  b_Crane$CraneSucked  THEN
                 b_Crane$_transit  := TRUE;
                 b_Crane$_state  := Crane_states_t#Step0;
            END_IF

        Crane_states_t#Crane_On_Conveyor:
             b_Crane$_transit  := FALSE;
             b_Crane$CraneTurnCounterclockwise  := FALSE;
             b_Crane$CraneTurnClockwise  := FALSE;
             b_Crane$CraneLower  := TRUE;
            IF  b_Crane$CraneDown  THEN
                 b_Crane$_transit  := TRUE;
                 b_Crane$_state  := Crane_states_t#release;
            END_IF

        Crane_states_t#Crane_On_Conveyor_Metallic:
             b_Crane$_transit  := FALSE;
             b_Crane$CraneTurnCounterclockwise  := FALSE;
             b_Crane$CraneTurnClockwise  := FALSE;
             b_Crane$CraneLower  := TRUE;
            IF  b_Crane$CraneDown  THEN
                 b_Crane$_transit  := TRUE;
                 b_Crane$_state  := Crane_states_t#release;
            END_IF

        Crane_states_t#Crane_On_Conveyor_Metallic2:
             b_Crane$_transit  := FALSE;
             b_Crane$CraneTurnCounterclockwise  := FALSE;
             b_Crane$CraneTurnClockwise  := FALSE;
             b_Crane$CraneLower  := TRUE;
            IF  b_Crane$CraneDown  THEN
                 b_Crane$_transit  := TRUE;
                 b_Crane$_state  := Crane_states_t#release2;
            END_IF

        Crane_states_t#Crane_On_Conveyor_Not_Metallica_Black:
             b_Crane$_transit  := FALSE;
             b_Crane$CraneTurnCounterclockwise  := FALSE;
             b_Crane$CraneTurnClockwise  := FALSE;
             b_Crane$CraneLower  := TRUE;
            IF  b_Crane$CraneDown  THEN
                 b_Crane$_transit  := TRUE;
                 b_Crane$_state  := Crane_states_t#release_Black;
            END_IF

        Crane_states_t#Crane_On_Stamp_Metallic:
             b_Crane$_transit  := FALSE;
             b_Crane$CraneTurnCounterclockwise  := FALSE;
             b_Crane$CraneTurnClockwise  := FALSE;
             b_Crane$CraneLower  := TRUE;
            IF  b_Crane$CraneDown  THEN
                 b_Crane$_transit  := TRUE;
                 b_Crane$_state  := Crane_states_t#release_Workpiece;
            END_IF

        Crane_states_t#Crane_On_Stamp_Metallic2:
             b_Crane$_transit  := FALSE;
             b_Crane$CraneTurnCounterclockwise  := FALSE;
             b_Crane$CraneTurnClockwise  := FALSE;
            IF  b_Crane$StampLowered  THEN
                 b_Crane$_transit  := TRUE;
                 b_Crane$_state  := Crane_states_t#Interstep_4;
            END_IF

        Crane_states_t#Crane_On_Stamp_Metallic2_Lower:
             b_Crane$_transit  := FALSE;
             b_Crane$CraneLower  := TRUE;
            IF  b_Crane$CraneDown  THEN
                 b_Crane$_transit  := TRUE;
                 b_Crane$_state  := Crane_states_t#Suck_At_Stamp2;
            END_IF

        Crane_states_t#Crane_On_Stamp_Stop_Black:
             b_Crane$_transit  := FALSE;
             b_Crane$CraneTurnClockwise  := FALSE;
             b_Crane$CraneTurnCounterclockwise  := FALSE;
            IF TRUE THEN
                 b_Crane$_transit  := TRUE;
                 b_Crane$_state  := Crane_states_t#Reset_interconnect;
            END_IF

        Crane_states_t#Crane_On_Stamp_White:
             b_Crane$_transit  := FALSE;
             b_Crane$CraneTurnCounterclockwise  := FALSE;
             b_Crane$CraneTurnClockwise  := FALSE;
             b_Crane$CraneLower  := TRUE;
            IF  b_Crane$CraneDown  THEN
                 b_Crane$_transit  := TRUE;
                 b_Crane$_state  := Crane_states_t#release_Workpiece_White;
            END_IF

        Crane_states_t#Crane_Turn_Left_Back_To_Stamp:
             b_Crane$_transit  := FALSE;
             b_Crane$CraneTurnCounterclockwise  := TRUE;
             b_Crane$CraneTurnClockwise  := FALSE;
            IF (( b_Crane$AnalogCranePosition  > INT#8160) AND ( b_Crane$AnalogCranePosition  < INT#8260)) THEN
                 b_Crane$_transit  := TRUE;
                 b_Crane$_state  := Crane_states_t#Crane_On_Stamp_Stop_Black;
            END_IF

        Crane_states_t#Crane_Turn_Left_From_Stamp:
             b_Crane$_transit  := FALSE;
             b_Crane$CraneTurnClockwise  := TRUE;
             b_Crane$CraneTurnCounterclockwise  := FALSE;
            IF (( b_Crane$AnalogCranePosition  > INT#16060) AND ( b_Crane$AnalogCranePosition  < INT#16160)) THEN
                 b_Crane$_transit  := TRUE;
                 b_Crane$_state  := Crane_states_t#Crane_On_Conveyor_Metallic;
            END_IF

        Crane_states_t#Crane_Turn_Left_Metallic:
             b_Crane$_transit  := FALSE;
             b_Crane$CraneTurnCounterclockwise  := TRUE;
             b_Crane$CraneTurnClockwise  := FALSE;
            IF (( b_Crane$AnalogCranePosition  > INT#8160) AND ( b_Crane$AnalogCranePosition  < INT#8260)) THEN
                 b_Crane$_transit  := TRUE;
                 b_Crane$_state  := Crane_states_t#Crane_On_Stamp_Metallic;
            END_IF

        Crane_states_t#Crane_Turn_Left_Metallic2:
             b_Crane$_transit  := FALSE;
             b_Crane$CraneTurnCounterclockwise  := TRUE;
             b_Crane$CraneTurnClockwise  := FALSE;
            IF (( b_Crane$AnalogCranePosition  > INT#8160) AND ( b_Crane$AnalogCranePosition  < INT#8260)) THEN
                 b_Crane$_transit  := TRUE;
                 b_Crane$_state  := Crane_states_t#Crane_On_Stamp_Metallic2;
            END_IF

        Crane_states_t#Crane_Turn_Left_NOT_Metallic:
             b_Crane$_transit  := FALSE;
             b_Crane$CraneTurnCounterclockwise  := TRUE;
             b_Crane$CraneTurnClockwise  := FALSE;
            IF (( b_Crane$AnalogCranePosition  > INT#16160) AND ( b_Crane$AnalogCranePosition  < INT#16260)) THEN
                 b_Crane$_transit  := TRUE;
                 b_Crane$_state  := Crane_states_t#Crane_On_Conveyor;
            END_IF

        Crane_states_t#Crane_Turn_Left_NOT_Metallic_Black:
             b_Crane$_transit  := FALSE;
             b_Crane$CraneTurnCounterclockwise  := TRUE;
             b_Crane$CraneTurnClockwise  := FALSE;
            IF (( b_Crane$AnalogCranePosition  > INT#16160) AND ( b_Crane$AnalogCranePosition  < INT#16260)) THEN
                 b_Crane$_transit  := TRUE;
                 b_Crane$_state  := Crane_states_t#Crane_On_Conveyor_Not_Metallica_Black;
            END_IF

        Crane_states_t#Crane_Turn_Left_White:
             b_Crane$_transit  := FALSE;
             b_Crane$CraneTurnCounterclockwise  := TRUE;
             b_Crane$CraneTurnClockwise  := FALSE;
            IF (( b_Crane$AnalogCranePosition  > INT#8160) AND ( b_Crane$AnalogCranePosition  < INT#8260)) THEN
                 b_Crane$_transit  := TRUE;
                 b_Crane$_state  := Crane_states_t#Crane_On_Stamp_White;
            END_IF

        Crane_states_t#Crane_Turn_Right_From_Stamp:
             b_Crane$_transit  := FALSE;
             b_Crane$CraneTurnClockwise  := TRUE;
             b_Crane$CraneTurnCounterclockwise  := FALSE;
            IF (( b_Crane$AnalogCranePosition  > INT#16160) AND ( b_Crane$AnalogCranePosition  < INT#16260)) THEN
                 b_Crane$_transit  := TRUE;
                 b_Crane$_state  := Crane_states_t#Crane_On_Conveyor_Metallic2;
            END_IF

        Crane_states_t#Init:
             b_Crane$_transit  := FALSE;
            IF TRUE THEN
                 b_Crane$_transit  := TRUE;
                 b_Crane$_state  := Crane_states_t#Start_Crane;
            END_IF

        Crane_states_t#Interstep:
             b_Crane$_transit  := FALSE;
             b_Crane$StartCommandCrane  := TRUE;
            IF  b_Crane$StartVar  THEN
                 b_Crane$_transit  := TRUE;
                 b_Crane$_state  := Crane_states_t#Interstep_2;
            END_IF

        Crane_states_t#Interstep_2:
             b_Crane$_transit  := FALSE;
            IF  b_Crane$SliderMovedOut  THEN
                 b_Crane$_transit  := TRUE;
                 b_Crane$_state  := Crane_states_t#TimeDelay;
            END_IF

        Crane_states_t#Interstep_3:
             b_Crane$_transit  := FALSE;
            IF NOT  b_Crane$WorkpieceReady  THEN
                 b_Crane$_transit  := TRUE;
                 b_Crane$_state  := Crane_states_t#No_Workpiece_ready;
            ELSEIF  b_Crane$WorkpieceReady  THEN
                 b_Crane$_transit  := TRUE;
                 b_Crane$_state  := Crane_states_t#Turn_Right;
            END_IF

        Crane_states_t#Interstep_4:
             b_Crane$_transit  := FALSE;
            IF  b_Crane$StampSliderSensorMovedOut  THEN
                 b_Crane$_transit  := TRUE;
                 b_Crane$_state  := Crane_states_t#Crane_On_Stamp_Metallic2_Lower;
            END_IF

        Crane_states_t#Lower_Crane:
             b_Crane$_transit  := FALSE;
             b_Crane$CraneLower  := TRUE;
            IF  b_Crane$CraneDown  THEN
                 b_Crane$_transit  := TRUE;
                 b_Crane$_state  := Crane_states_t#Suck_At_Stamp;
            END_IF

        Crane_states_t#Magazin_Stop:
             b_Crane$_transit  := FALSE;
             b_Crane$CraneTurnClockwise  := FALSE;
             b_Crane$CraneTurnCounterclockwise  := FALSE;
            IF TRUE THEN
                 b_Crane$_transit  := TRUE;
                 b_Crane$_state  := Crane_states_t#Crane_Lower;
            END_IF

        Crane_states_t#Magazin_Stop_Black:
             b_Crane$_transit  := FALSE;
             b_Crane$CraneTurnClockwise  := FALSE;
             b_Crane$CraneTurnCounterclockwise  := FALSE;
             b_Crane$MagazinVacuumOn  := TRUE;
             b_Crane$MagazinVacuumOff  := FALSE;
             b_Crane$CraneLower  := TRUE;
            IF  b_Crane$CraneSucked  THEN
                 b_Crane$_transit  := TRUE;
                 b_Crane$_state  := Crane_states_t#Crane_Lift_NOT_Metallic_Black;
            END_IF

        Crane_states_t#Magazin_Stop_Final:
             b_Crane$_transit  := FALSE;
             b_Crane$CraneTurnClockwise  := FALSE;
             b_Crane$CraneTurnCounterclockwise  := FALSE;
            IF TRUE THEN
                 b_Crane$_transit  := TRUE;
                 b_Crane$_state  := Crane_states_t#Start_Crane;
            END_IF

        Crane_states_t#No_Workpiece_ready:
             b_Crane$_transit  := FALSE;
             b_Crane$MagazinVacuumOn  := FALSE;
             b_Crane$MagazinVacuumOff  := FALSE;
             b_Crane$CraneLower  := FALSE;
            IF  b_Crane$StampSliderFilled  THEN
                 b_Crane$_transit  := TRUE;
                 b_Crane$_state  := Crane_states_t#Crane_Turn_Left_Metallic2;
            ELSEIF NOT  b_Crane$StampSliderFilled  THEN
                 b_Crane$_transit  := TRUE;
                 b_Crane$_state  := Crane_states_t#Turn_Right_Final;
            END_IF

        Crane_states_t#Reset_interconnect:
             b_Crane$_transit  := FALSE;
             b_Crane$interconnect  := FALSE;
             b_Crane$Timer1$IN  := FALSE;
             b_Crane$Timer1$PT  := USINT#0;
            IF  b_Crane$Timer1$IN  THEN
                 b_Crane$Timer1$Q  := ( b_Crane$Timer1$ET  = USINT#0);
                IF ( b_Crane$Timer1$ET  > USINT#0) THEN
                     b_Crane$Timer1$ET  := ( b_Crane$Timer1$ET  - USINT#1);
                ELSE
                     b_Crane$Timer1$ET  := USINT#0;
                END_IF
            ELSE
                 b_Crane$Timer1$Q  := FALSE;
                 b_Crane$Timer1$ET  :=  b_Crane$Timer1$PT ;
            END_IF
            IF  b_Crane$SliderMovedOut  THEN
                 b_Crane$_transit  := TRUE;
                 b_Crane$_state  := Crane_states_t#Lower_Crane;
            END_IF

        Crane_states_t#Stamp_Pressure_Profile_Set_Metallic:
             b_Crane$_transit  := FALSE;
             b_Crane$AnalogCranePressure  :=  b_PARAMETER_CRANE_PRESSURE_METALLIC ;
            IF TRUE THEN
                 b_Crane$_transit  := TRUE;
                 b_Crane$_state  := Crane_states_t#Crane_Lift_Magazin_Metallic;
            END_IF

        Crane_states_t#Stamp_Pressure_Profile_Set_White:
             b_Crane$_transit  := FALSE;
             b_Crane$AnalogCranePressure  :=  b_PARAMETER_CRANE_PRESSURE_WHITE ;
            IF TRUE THEN
                 b_Crane$_transit  := TRUE;
                 b_Crane$_state  := Crane_states_t#Crane_Lift_Magazin_White;
            END_IF

        Crane_states_t#Start_Crane:
             b_Crane$_transit  := FALSE;
             b_Crane$CraneLower  := FALSE;
             b_Crane$MagazinVacuumOff  := FALSE;
             b_Crane$MagazinVacuumOn  := FALSE;
             b_Crane$CraneTurnCounterclockwise  := FALSE;
             b_Crane$CraneTurnClockwise  := FALSE;
             b_Crane$AnalogCranePressure  := INT#0;
             b_Crane$StartVar  := FALSE;
             b_Crane$StartCommandCrane  := FALSE;
            IF ( b_Crane$StartButtonMagazin  = TRUE) THEN
                 b_Crane$interconnectCraneStartCommand  := TRUE;
            END_IF
            IF  b_Crane$interconnectCraneStartCommand  THEN
                 b_Crane$_transit  := TRUE;
                 b_Crane$_state  := Crane_states_t#Crane_Init;
            END_IF

        Crane_states_t#Step0:
             b_Crane$_transit  := FALSE;
            IF ( b_Crane$MagazinCapacitiveSensor  AND  b_Crane$MagazinOpticalSensor ) THEN
                 b_Crane$_transit  := TRUE;
                 b_Crane$_state  := Crane_states_t#Stamp_Pressure_Profile_Set_Metallic;
            ELSEIF (NOT  b_Crane$MagazinCapacitiveSensor  AND  b_Crane$MagazinOpticalSensor ) THEN
                 b_Crane$_transit  := TRUE;
                 b_Crane$_state  := Crane_states_t#Stamp_Pressure_Profile_Set_White;
            ELSEIF (NOT  b_Crane$MagazinCapacitiveSensor  AND NOT  b_Crane$MagazinOpticalSensor ) THEN
                 b_Crane$_transit  := TRUE;
                 b_Crane$_state  := Crane_states_t#Crane_Lift_Magazin;
            END_IF

        Crane_states_t#Step2:
             b_Crane$_transit  := FALSE;
            IF ( b_Crane$MagazinCapacitiveSensor  OR  b_Crane$MagazinOpticalSensor ) THEN
                 b_Crane$_transit  := TRUE;
                 b_Crane$_state  := Crane_states_t#pause;
            ELSEIF (NOT  b_Crane$MagazinCapacitiveSensor  AND NOT  b_Crane$MagazinOpticalSensor ) THEN
                 b_Crane$_transit  := TRUE;
                 b_Crane$_state  := Crane_states_t#Turn_Right_Black;
            END_IF

        Crane_states_t#Step3:
             b_Crane$_transit  := FALSE;
            IF NOT  b_Crane$WorkpieceReady  THEN
                 b_Crane$_transit  := TRUE;
                 b_Crane$_state  := Crane_states_t#Step4;
            ELSEIF  b_Crane$WorkpieceReady  THEN
                 b_Crane$_transit  := TRUE;
                 b_Crane$_state  := Crane_states_t#Step2;
            END_IF

        Crane_states_t#Step4:
             b_Crane$_transit  := FALSE;
            IF TRUE THEN
                 b_Crane$_transit  := TRUE;
                 b_Crane$_state  := Crane_states_t#Interstep;
            END_IF

        Crane_states_t#Suck_At_Stamp:
             b_Crane$_transit  := FALSE;
             b_Crane$MagazinVacuumOn  := TRUE;
             b_Crane$MagazinVacuumOff  := FALSE;
            IF  b_Crane$CraneSucked  THEN
                 b_Crane$_transit  := TRUE;
                 b_Crane$_state  := Crane_states_t#Crane_Lift_At_Stamp;
            END_IF

        Crane_states_t#Suck_At_Stamp2:
             b_Crane$_transit  := FALSE;
             b_Crane$MagazinVacuumOn  := TRUE;
             b_Crane$MagazinVacuumOff  := FALSE;
            IF  b_Crane$CraneSucked  THEN
                 b_Crane$_transit  := TRUE;
                 b_Crane$_state  := Crane_states_t#Crane_Lift_At_Stamp2;
            END_IF

        Crane_states_t#TimeDelay:
             b_Crane$_transit  := FALSE;
             b_Crane$TimeDelay_Timer$IN  := TRUE;
             b_Crane$TimeDelay_Timer$PT  :=  b_Crane$TimeDelay_Timer_Duration ;
            IF  b_Crane$TimeDelay_Timer$IN  THEN
                 b_Crane$TimeDelay_Timer$Q  := ( b_Crane$TimeDelay_Timer$ET  = USINT#0);
                IF ( b_Crane$TimeDelay_Timer$ET  > USINT#0) THEN
                     b_Crane$TimeDelay_Timer$ET  := ( b_Crane$TimeDelay_Timer$ET  - USINT#1);
                ELSE
                     b_Crane$TimeDelay_Timer$ET  := USINT#0;
                END_IF
            ELSE
                 b_Crane$TimeDelay_Timer$Q  := FALSE;
                 b_Crane$TimeDelay_Timer$ET  :=  b_Crane$TimeDelay_Timer$PT ;
            END_IF
             b_Crane$TimeDelay_Timer_interconnect  :=  b_Crane$TimeDelay_Timer$Q ;
            IF  b_Crane$TimeDelay_Timer_interconnect  THEN
                 b_Crane$_transit  := TRUE;
                 b_Crane$_state  := Crane_states_t#Interstep_3;
            END_IF

        Crane_states_t#Turn_Right:
             b_Crane$_transit  := FALSE;
             b_Crane$CraneTurnClockwise  := TRUE;
             b_Crane$CraneTurnCounterclockwise  := FALSE;
            IF (( b_Crane$AnalogCranePosition  > INT#24290) AND ( b_Crane$AnalogCranePosition  < INT#24390)) THEN
                 b_Crane$_transit  := TRUE;
                 b_Crane$_state  := Crane_states_t#Magazin_Stop;
            END_IF

        Crane_states_t#Turn_Right_Black:
             b_Crane$_transit  := FALSE;
             b_Crane$CraneTurnClockwise  := TRUE;
             b_Crane$CraneTurnCounterclockwise  := FALSE;
            IF (( b_Crane$AnalogCranePosition  > INT#24290) AND ( b_Crane$AnalogCranePosition  < INT#24390)) THEN
                 b_Crane$_transit  := TRUE;
                 b_Crane$_state  := Crane_states_t#Magazin_Stop_Black;
            END_IF

        Crane_states_t#Turn_Right_Final:
             b_Crane$_transit  := FALSE;
             b_Crane$CraneTurnClockwise  := TRUE;
             b_Crane$CraneTurnCounterclockwise  := FALSE;
             b_Crane$AnalogCranePressure  := INT#0;
            IF (( b_Crane$AnalogCranePosition  > INT#24290) AND ( b_Crane$AnalogCranePosition  < INT#24390)) THEN
                 b_Crane$_transit  := TRUE;
                 b_Crane$_state  := Crane_states_t#Magazin_Stop_Final;
            END_IF

        Crane_states_t#pause:
             b_Crane$_transit  := FALSE;
             b_Crane$Timer1$IN  :=  b_Crane$CraneUp ;
             b_Crane$Timer1$PT  :=  b_Crane$Duration1 ;
            IF  b_Crane$Timer1$IN  THEN
                 b_Crane$Timer1$Q  := ( b_Crane$Timer1$ET  = USINT#0);
                IF ( b_Crane$Timer1$ET  > USINT#0) THEN
                     b_Crane$Timer1$ET  := ( b_Crane$Timer1$ET  - USINT#1);
                ELSE
                     b_Crane$Timer1$ET  := USINT#0;
                END_IF
            ELSE
                 b_Crane$Timer1$Q  := FALSE;
                 b_Crane$Timer1$ET  :=  b_Crane$Timer1$PT ;
            END_IF
             b_Crane$interconnect  :=  b_Crane$Timer1$Q ;
            IF  b_Crane$interconnect  THEN
                 b_Crane$_transit  := TRUE;
                 b_Crane$_state  := Crane_states_t#Reset_interconnect;
            END_IF

        Crane_states_t#release:
             b_Crane$_transit  := FALSE;
             b_Crane$MagazinVacuumOff  := TRUE;
             b_Crane$MagazinVacuumOn  := FALSE;
            IF TRUE THEN
                 b_Crane$_transit  := TRUE;
                 b_Crane$_state  := Crane_states_t#Crane_Lift_Conveyor;
            END_IF

        Crane_states_t#release2:
             b_Crane$_transit  := FALSE;
             b_Crane$MagazinVacuumOff  := TRUE;
             b_Crane$MagazinVacuumOn  := FALSE;
            IF TRUE THEN
                 b_Crane$_transit  := TRUE;
                 b_Crane$_state  := Crane_states_t#Crane_Lift_Conveyor2;
            END_IF

        Crane_states_t#release_Black:
             b_Crane$_transit  := FALSE;
             b_Crane$MagazinVacuumOn  := FALSE;
             b_Crane$MagazinVacuumOff  := TRUE;
            IF TRUE THEN
                 b_Crane$_transit  := TRUE;
                 b_Crane$_state  := Crane_states_t#Crane_Lift_Conveyor_Black;
            END_IF

        Crane_states_t#release_Workpiece:
             b_Crane$_transit  := FALSE;
             b_Crane$MagazinVacuumOff  := TRUE;
             b_Crane$MagazinVacuumOn  := FALSE;
            IF TRUE THEN
                 b_Crane$_transit  := TRUE;
                 b_Crane$_state  := Crane_states_t#Crane_Go_Up;
            END_IF

        Crane_states_t#release_Workpiece_White:
             b_Crane$_transit  := FALSE;
             b_Crane$MagazinVacuumOff  := TRUE;
             b_Crane$MagazinVacuumOn  := FALSE;
            IF TRUE THEN
                 b_Crane$_transit  := TRUE;
                 b_Crane$_state  := Crane_states_t#Crane_Go_Up_White;
            END_IF

            END_CASE
    CASE  b_Stamp$_state  OF
        Stamp_states_t#Green_Lamp:
             b_Stamp$_transit  := FALSE;
             b_Stamp$StampGreenLamp  := TRUE;
             b_Stamp$interconnectStampStartCommand  := FALSE;
            IF TRUE THEN
                 b_Stamp$_transit  := TRUE;
                 b_Stamp$_state  := Stamp_states_t#Stamp_Init_1;
            END_IF

        Stamp_states_t#Init:
             b_Stamp$_transit  := FALSE;
            IF TRUE THEN
                 b_Stamp$_transit  := TRUE;
                 b_Stamp$_state  := Stamp_states_t#Start_Stamp;
            END_IF

        Stamp_states_t#Interstep:
             b_Stamp$_transit  := FALSE;
             b_Stamp$StartCommandStamp  := TRUE;
            IF  b_Stamp$StartVar  THEN
                 b_Stamp$_transit  := TRUE;
                 b_Stamp$_state  := Stamp_states_t#Intertsep_2;
            END_IF

        Stamp_states_t#Intertsep_2:
             b_Stamp$_transit  := FALSE;
            IF  b_Stamp$StampSliderFilled  THEN
                 b_Stamp$_transit  := TRUE;
                 b_Stamp$_state  := Stamp_states_t#Step0;
            END_IF

        Stamp_states_t#StampProcess:
             b_Stamp$_transit  := FALSE;
             b_Stamp$StampSliderMovedIn  := FALSE;
             b_Stamp$StampPusher  := TRUE;
            IF  b_Stamp$StampLowered  THEN
                 b_Stamp$_transit  := TRUE;
                 b_Stamp$_state  := Stamp_states_t#Step1;
            END_IF

        Stamp_states_t#StampSliderBack:
             b_Stamp$_transit  := FALSE;
             b_Stamp$StampSliderMovedIn  := TRUE;
             b_Stamp$StampSliderMovedOut  := FALSE;
            IF  b_Stamp$StampSliderSensorMovedIn  THEN
                 b_Stamp$_transit  := TRUE;
                 b_Stamp$_state  := Stamp_states_t#StampProcess;
            END_IF

        Stamp_states_t#StampSliderForward:
             b_Stamp$_transit  := FALSE;
             b_Stamp$StampPusher  := FALSE;
             b_Stamp$StampSliderMovedOut  := TRUE;
            IF (( b_Stamp$StampLowered  = FALSE) AND ( b_Stamp$StampUp  = TRUE)) THEN
                 b_Stamp$interconnect  := FALSE;
            END_IF
             b_Stamp$Timer$IN  := FALSE;
             b_Stamp$Timer$PT  := USINT#0;
            IF  b_Stamp$Timer$IN  THEN
                 b_Stamp$Timer$Q  := ( b_Stamp$Timer$ET  = USINT#0);
                IF ( b_Stamp$Timer$ET  > USINT#0) THEN
                     b_Stamp$Timer$ET  := ( b_Stamp$Timer$ET  - USINT#1);
                ELSE
                     b_Stamp$Timer$ET  := USINT#0;
                END_IF
            ELSE
                 b_Stamp$Timer$Q  := FALSE;
                 b_Stamp$Timer$ET  :=  b_Stamp$Timer$PT ;
            END_IF
            IF  b_Stamp$StampSliderMovedOut  THEN
                 b_Stamp$_transit  := TRUE;
                 b_Stamp$_state  := Stamp_states_t#Step2;
            END_IF

        Stamp_states_t#Stamp_Init_1:
             b_Stamp$_transit  := FALSE;
             b_Stamp$StampSliderMovedIn  := TRUE;
             b_Stamp$StampSliderMovedOut  := FALSE;
            IF  b_Stamp$StampSliderSensorMovedIn  THEN
                 b_Stamp$_transit  := TRUE;
                 b_Stamp$_state  := Stamp_states_t#Stamp_Init_2;
            END_IF

        Stamp_states_t#Stamp_Init_2:
             b_Stamp$_transit  := FALSE;
             b_Stamp$StampSliderMovedIn  := FALSE;
             b_Stamp$StampSliderMovedOut  := TRUE;
            IF  b_Stamp$StampSliderSensorMovedOut  THEN
                 b_Stamp$_transit  := TRUE;
                 b_Stamp$_state  := Stamp_states_t#Stamp_Init_3;
            END_IF

        Stamp_states_t#Stamp_Init_3:
             b_Stamp$_transit  := FALSE;
             b_Stamp$StampPusher  := TRUE;
            IF  b_Stamp$StampLowered  THEN
                 b_Stamp$_transit  := TRUE;
                 b_Stamp$_state  := Stamp_states_t#Stamp_Init_4;
            END_IF

        Stamp_states_t#Stamp_Init_4:
             b_Stamp$_transit  := FALSE;
             b_Stamp$StampPusher  := FALSE;
            IF  b_Stamp$StampUp  THEN
                 b_Stamp$_transit  := TRUE;
                 b_Stamp$_state  := Stamp_states_t#Interstep;
            END_IF

        Stamp_states_t#Start_Stamp:
             b_Stamp$_transit  := FALSE;
             b_Stamp$StampSliderMovedOut  := FALSE;
             b_Stamp$StampSliderMovedIn  := FALSE;
             b_Stamp$StampPusher  := FALSE;
             b_Stamp$StampGreenLamp  := FALSE;
             b_Stamp$StampPressure  := FALSE;
             b_Stamp$StartCommandStamp  := FALSE;
            IF ( b_Stamp$StampStartButton  = TRUE) THEN
                 b_Stamp$interconnectStampStartCommand  := TRUE;
            END_IF
            IF  b_Stamp$interconnectStampStartCommand  THEN
                 b_Stamp$_transit  := TRUE;
                 b_Stamp$_state  := Stamp_states_t#Green_Lamp;
            END_IF

        Stamp_states_t#Step0:
             b_Stamp$_transit  := FALSE;
            IF  b_Stamp$CraneUp  THEN
                 b_Stamp$_transit  := TRUE;
                 b_Stamp$_state  := Stamp_states_t#StampSliderBack;
            END_IF

        Stamp_states_t#Step1:
             b_Stamp$_transit  := FALSE;
             b_Stamp$Timer$IN  :=  b_Stamp$StampLowered ;
             b_Stamp$Timer$PT  := USINT#0;
            IF  b_Stamp$Timer$IN  THEN
                 b_Stamp$Timer$Q  := ( b_Stamp$Timer$ET  = USINT#0);
                IF ( b_Stamp$Timer$ET  > USINT#0) THEN
                     b_Stamp$Timer$ET  := ( b_Stamp$Timer$ET  - USINT#1);
                ELSE
                     b_Stamp$Timer$ET  := USINT#0;
                END_IF
            ELSE
                 b_Stamp$Timer$Q  := FALSE;
                 b_Stamp$Timer$ET  :=  b_Stamp$Timer$PT ;
            END_IF
             b_Stamp$interconnect  :=  b_Stamp$Timer$Q ;
            IF  b_Stamp$interconnect  THEN
                 b_Stamp$_transit  := TRUE;
                 b_Stamp$_state  := Stamp_states_t#StampSliderForward;
            END_IF

        Stamp_states_t#Step2:
             b_Stamp$_transit  := FALSE;
            IF ((( b_Stamp$AnalogCranePosition  > INT#16160) AND ( b_Stamp$AnalogCranePosition  < INT#16260)) AND NOT  b_Stamp$StampSliderFilled ) THEN
                 b_Stamp$_transit  := TRUE;
                 b_Stamp$_state  := Stamp_states_t#Interstep;
            END_IF

            END_CASE
    CASE  b_Conveyor$_state  OF
        Conveyor_states_t#Conveyor_Init:
             b_Conveyor$_transit  := FALSE;
             b_Conveyor$SorterConveyorTowardsStacker  := TRUE;
             b_Conveyor$SorterConveyorTowardsCrane  := FALSE;
             b_Conveyor$Timer_Conveyor_Test$IN  := TRUE;
             b_Conveyor$Timer_Conveyor_Test$PT  :=  b_Conveyor$Duration_Conveyor_Test ;
            IF  b_Conveyor$Timer_Conveyor_Test$IN  THEN
                 b_Conveyor$Timer_Conveyor_Test$Q  := ( b_Conveyor$Timer_Conveyor_Test$ET  = USINT#0);
                IF ( b_Conveyor$Timer_Conveyor_Test$ET  > USINT#0) THEN
                     b_Conveyor$Timer_Conveyor_Test$ET  := ( b_Conveyor$Timer_Conveyor_Test$ET  - USINT#1);
                ELSE
                     b_Conveyor$Timer_Conveyor_Test$ET  := USINT#0;
                END_IF
            ELSE
                 b_Conveyor$Timer_Conveyor_Test$Q  := FALSE;
                 b_Conveyor$Timer_Conveyor_Test$ET  :=  b_Conveyor$Timer_Conveyor_Test$PT ;
            END_IF
             b_Conveyor$interconnect_Conveyor_Test  :=  b_Conveyor$Timer_Conveyor_Test$Q ;
            IF  b_Conveyor$interconnect_Conveyor_Test  THEN
                 b_Conveyor$_transit  := TRUE;
                 b_Conveyor$_state  := Conveyor_states_t#Conveyor_init_2;
            END_IF

        Conveyor_states_t#Conveyor_Stop_Empty_Magazin:
             b_Conveyor$_transit  := FALSE;
             b_Conveyor$SorterConveyorTowardsStacker  := FALSE;
             b_Conveyor$SorterConveyorTowardsCrane  := FALSE;
             b_Conveyor$interconnectConveyorStartCommand  := FALSE;
            IF TRUE THEN
                 b_Conveyor$_transit  := TRUE;
                 b_Conveyor$_state  := Conveyor_states_t#Interstep;
            END_IF

        Conveyor_states_t#Conveyor_Towards_Stacker:
             b_Conveyor$_transit  := FALSE;
             b_Conveyor$SorterConveyorTowardsStacker  := TRUE;
             b_Conveyor$SorterConveyorTowardsCrane  := FALSE;
            IF TRUE THEN
                 b_Conveyor$_transit  := TRUE;
                 b_Conveyor$_state  := Conveyor_states_t#Runtime_Conveyor;
            END_IF

        Conveyor_states_t#Conveyor_init_2:
             b_Conveyor$_transit  := FALSE;
             b_Conveyor$SorterConveyorTowardsStacker  := FALSE;
             b_Conveyor$SorterConveyorTowardsCrane  := FALSE;
             b_Conveyor$interconnect_Conveyor_Test  := FALSE;
             b_Conveyor$Timer_Conveyor_Test$IN  := FALSE;
             b_Conveyor$Timer_Conveyor_Test$PT  := USINT#0;
            IF  b_Conveyor$Timer_Conveyor_Test$IN  THEN
                 b_Conveyor$Timer_Conveyor_Test$Q  := ( b_Conveyor$Timer_Conveyor_Test$ET  = USINT#0);
                IF ( b_Conveyor$Timer_Conveyor_Test$ET  > USINT#0) THEN
                     b_Conveyor$Timer_Conveyor_Test$ET  := ( b_Conveyor$Timer_Conveyor_Test$ET  - USINT#1);
                ELSE
                     b_Conveyor$Timer_Conveyor_Test$ET  := USINT#0;
                END_IF
            ELSE
                 b_Conveyor$Timer_Conveyor_Test$Q  := FALSE;
                 b_Conveyor$Timer_Conveyor_Test$ET  :=  b_Conveyor$Timer_Conveyor_Test$PT ;
            END_IF
            IF TRUE THEN
                 b_Conveyor$_transit  := TRUE;
                 b_Conveyor$_state  := Conveyor_states_t#Interstep;
            END_IF

        Conveyor_states_t#Conveyor_pause:
             b_Conveyor$_transit  := FALSE;
             b_Conveyor$SorterConveyorTowardsStacker  := FALSE;
             b_Conveyor$SorterConveyorTowardsCrane  := FALSE;
             b_Conveyor$interconnect_Conveyor_Runtime  := FALSE;
             b_Conveyor$Timer_Conveyor_Runtime$IN  := FALSE;
             b_Conveyor$Timer_Conveyor_Runtime$PT  := USINT#0;
            IF  b_Conveyor$Timer_Conveyor_Runtime$IN  THEN
                 b_Conveyor$Timer_Conveyor_Runtime$Q  := ( b_Conveyor$Timer_Conveyor_Runtime$ET  = USINT#0);
                IF ( b_Conveyor$Timer_Conveyor_Runtime$ET  > USINT#0) THEN
                     b_Conveyor$Timer_Conveyor_Runtime$ET  := ( b_Conveyor$Timer_Conveyor_Runtime$ET  - USINT#1);
                ELSE
                     b_Conveyor$Timer_Conveyor_Runtime$ET  := USINT#0;
                END_IF
            ELSE
                 b_Conveyor$Timer_Conveyor_Runtime$Q  := FALSE;
                 b_Conveyor$Timer_Conveyor_Runtime$ET  :=  b_Conveyor$Timer_Conveyor_Runtime$PT ;
            END_IF
            IF TRUE THEN
                 b_Conveyor$_transit  := TRUE;
                 b_Conveyor$_state  := Conveyor_states_t#Interstep;
            END_IF

        Conveyor_states_t#Green_Lamp:
             b_Conveyor$_transit  := FALSE;
             b_Conveyor$SorterGreenLampConveyor  := TRUE;
             b_Conveyor$interconnectConveyorStartCommand  := FALSE;
            IF TRUE THEN
                 b_Conveyor$_transit  := TRUE;
                 b_Conveyor$_state  := Conveyor_states_t#Conveyor_Init;
            END_IF

        Conveyor_states_t#Init:
             b_Conveyor$_transit  := FALSE;
            IF TRUE THEN
                 b_Conveyor$_transit  := TRUE;
                 b_Conveyor$_state  := Conveyor_states_t#Start_Conveyor;
            END_IF

        Conveyor_states_t#Interstep:
             b_Conveyor$_transit  := FALSE;
             b_Conveyor$StartCommandConveyor  := TRUE;
            IF  b_Conveyor$StartVar  THEN
                 b_Conveyor$_transit  := TRUE;
                 b_Conveyor$_state  := Conveyor_states_t#Step0;
            END_IF

        Conveyor_states_t#Runtime_Conveyor:
             b_Conveyor$_transit  := FALSE;
             b_Conveyor$Timer_Conveyor_Runtime$IN  := TRUE;
             b_Conveyor$Timer_Conveyor_Runtime$PT  :=  b_Conveyor$Duration_Conveyor_Runtime ;
            IF  b_Conveyor$Timer_Conveyor_Runtime$IN  THEN
                 b_Conveyor$Timer_Conveyor_Runtime$Q  := ( b_Conveyor$Timer_Conveyor_Runtime$ET  = USINT#0);
                IF ( b_Conveyor$Timer_Conveyor_Runtime$ET  > USINT#0) THEN
                     b_Conveyor$Timer_Conveyor_Runtime$ET  := ( b_Conveyor$Timer_Conveyor_Runtime$ET  - USINT#1);
                ELSE
                     b_Conveyor$Timer_Conveyor_Runtime$ET  := USINT#0;
                END_IF
            ELSE
                 b_Conveyor$Timer_Conveyor_Runtime$Q  := FALSE;
                 b_Conveyor$Timer_Conveyor_Runtime$ET  :=  b_Conveyor$Timer_Conveyor_Runtime$PT ;
            END_IF
             b_Conveyor$interconnect_Conveyor_Runtime  :=  b_Conveyor$Timer_Conveyor_Runtime$Q ;
            IF  b_Conveyor$interconnect_Conveyor_Runtime  THEN
                 b_Conveyor$_transit  := TRUE;
                 b_Conveyor$_state  := Conveyor_states_t#Conveyor_pause;
            END_IF

        Conveyor_states_t#Start_Conveyor:
             b_Conveyor$_transit  := FALSE;
             b_Conveyor$interconnectConveyorTerminationCommand  := FALSE;
             b_Conveyor$SorterConveyorTowardsStacker  := FALSE;
             b_Conveyor$SorterConveyorTowardsCrane  := FALSE;
             b_Conveyor$SorterGreenLampConveyor  := FALSE;
             b_Conveyor$interconnect_Conveyor_Runtime  := FALSE;
             b_Conveyor$interconnect_Conveyor_Test  := FALSE;
             b_Conveyor$Timer_Conveyor_Test$IN  := FALSE;
             b_Conveyor$Timer_Conveyor_Test$PT  := USINT#0;
            IF  b_Conveyor$Timer_Conveyor_Test$IN  THEN
                 b_Conveyor$Timer_Conveyor_Test$Q  := ( b_Conveyor$Timer_Conveyor_Test$ET  = USINT#0);
                IF ( b_Conveyor$Timer_Conveyor_Test$ET  > USINT#0) THEN
                     b_Conveyor$Timer_Conveyor_Test$ET  := ( b_Conveyor$Timer_Conveyor_Test$ET  - USINT#1);
                ELSE
                     b_Conveyor$Timer_Conveyor_Test$ET  := USINT#0;
                END_IF
            ELSE
                 b_Conveyor$Timer_Conveyor_Test$Q  := FALSE;
                 b_Conveyor$Timer_Conveyor_Test$ET  :=  b_Conveyor$Timer_Conveyor_Test$PT ;
            END_IF
             b_Conveyor$Timer_Conveyor_Runtime$IN  := FALSE;
             b_Conveyor$Timer_Conveyor_Runtime$PT  := USINT#0;
            IF  b_Conveyor$Timer_Conveyor_Runtime$IN  THEN
                 b_Conveyor$Timer_Conveyor_Runtime$Q  := ( b_Conveyor$Timer_Conveyor_Runtime$ET  = USINT#0);
                IF ( b_Conveyor$Timer_Conveyor_Runtime$ET  > USINT#0) THEN
                     b_Conveyor$Timer_Conveyor_Runtime$ET  := ( b_Conveyor$Timer_Conveyor_Runtime$ET  - USINT#1);
                ELSE
                     b_Conveyor$Timer_Conveyor_Runtime$ET  := USINT#0;
                END_IF
            ELSE
                 b_Conveyor$Timer_Conveyor_Runtime$Q  := FALSE;
                 b_Conveyor$Timer_Conveyor_Runtime$ET  :=  b_Conveyor$Timer_Conveyor_Runtime$PT ;
            END_IF
             b_Conveyor$StartVar  := FALSE;
             b_Conveyor$StartCommandConveyor  := FALSE;
            IF ( b_Conveyor$SorterStartButton  = TRUE) THEN
                 b_Conveyor$interconnectConveyorStartCommand  := TRUE;
            END_IF
            IF  b_Conveyor$interconnectConveyorStartCommand  THEN
                 b_Conveyor$_transit  := TRUE;
                 b_Conveyor$_state  := Conveyor_states_t#Green_Lamp;
            END_IF

        Conveyor_states_t#Step0:
             b_Conveyor$_transit  := FALSE;
            IF  b_Conveyor$SorterLightbarrierCraneInterface  THEN
                 b_Conveyor$_transit  := TRUE;
                 b_Conveyor$_state  := Conveyor_states_t#Conveyor_Towards_Stacker;
            ELSEIF NOT  b_Conveyor$SorterLightbarrierCraneInterface  THEN
                 b_Conveyor$_transit  := TRUE;
                 b_Conveyor$_state  := Conveyor_states_t#Conveyor_Stop_Empty_Magazin;
            END_IF

            END_CASE
    CASE  b_Pusher$_state  OF
        Pusher_states_t#Check_For_Black:
             b_Pusher$_transit  := FALSE;
            IF (( b_Pusher$Slide2_black  = INT#1) AND ( b_Pusher$Priority_Var_Black  = INT#2)) THEN
                 b_Pusher$_transit  := TRUE;
                 b_Pusher$_state  := Pusher_states_t#Second_Slide_black_workpieces;
            ELSEIF (( b_Pusher$Slide3_black  = INT#1) AND ( b_Pusher$Priority_Var_Black  = INT#3)) THEN
                 b_Pusher$_transit  := TRUE;
                 b_Pusher$_state  := Pusher_states_t#Third_Slide_black_workpieces;
            ELSEIF (( b_Pusher$Slide1_black  = INT#1) AND ( b_Pusher$Priority_Var_Black  = INT#1)) THEN
                 b_Pusher$_transit  := TRUE;
                 b_Pusher$_state  := Pusher_states_t#First_Slide_black_workpieces;
            END_IF

        Pusher_states_t#Check_For_Metal:
             b_Pusher$_transit  := FALSE;
            IF (( b_Pusher$Slide3_metal  = INT#1) AND ( b_Pusher$Priority_Var_Metal  = INT#3)) THEN
                 b_Pusher$_transit  := TRUE;
                 b_Pusher$_state  := Pusher_states_t#Third_Slide_metal_workpieces;
            ELSEIF (( b_Pusher$Slide2_metal  = INT#1) AND ( b_Pusher$Priority_Var_Metal  = INT#2)) THEN
                 b_Pusher$_transit  := TRUE;
                 b_Pusher$_state  := Pusher_states_t#Second_Slide_metal_workpieces;
            ELSEIF (( b_Pusher$Slide1_metal  = INT#1) AND ( b_Pusher$Priority_Var_Metal  = INT#1)) THEN
                 b_Pusher$_transit  := TRUE;
                 b_Pusher$_state  := Pusher_states_t#First_Slide_metal_workpieces;
            END_IF

        Pusher_states_t#Check_For_White:
             b_Pusher$_transit  := FALSE;
            IF (( b_Pusher$Slide1_white  = INT#1) AND ( b_Pusher$Priority_Var_White  = INT#1)) THEN
                 b_Pusher$_transit  := TRUE;
                 b_Pusher$_state  := Pusher_states_t#First_Slide_white_workpieces;
            ELSEIF (( b_Pusher$Slide3_white  = INT#1) AND ( b_Pusher$Priority_Var_White  = INT#3)) THEN
                 b_Pusher$_transit  := TRUE;
                 b_Pusher$_state  := Pusher_states_t#Third_Slide_white_workpieces;
            ELSEIF (( b_Pusher$Slide2_white  = INT#1) AND ( b_Pusher$Priority_Var_White  = INT#2)) THEN
                 b_Pusher$_transit  := TRUE;
                 b_Pusher$_state  := Pusher_states_t#Second_Slide_white_workpieces;
            END_IF

        Pusher_states_t#First_Slide_Timer_Black:
             b_Pusher$_transit  := FALSE;
            IF ( b_Pusher$SorterLightnesssensorCraneInterfaceInverse  = TRUE) THEN
                 b_Pusher$Timer_Slide1_Black$IN  :=  b_Pusher$SorterLightnesssensorCraneInterfaceInverse ;
                 b_Pusher$Timer_Slide1_Black$PT  :=  b_Pusher$Duration_Slide1_Black ;
                IF  b_Pusher$Timer_Slide1_Black$IN  THEN
                     b_Pusher$Timer_Slide1_Black$Q  := ( b_Pusher$Timer_Slide1_Black$ET  = USINT#0);
                    IF ( b_Pusher$Timer_Slide1_Black$ET  > USINT#0) THEN
                         b_Pusher$Timer_Slide1_Black$ET  := ( b_Pusher$Timer_Slide1_Black$ET  - USINT#1);
                    ELSE
                         b_Pusher$Timer_Slide1_Black$ET  := USINT#0;
                    END_IF
                ELSE
                     b_Pusher$Timer_Slide1_Black$Q  := FALSE;
                     b_Pusher$Timer_Slide1_Black$ET  :=  b_Pusher$Timer_Slide1_Black$PT ;
                END_IF
                 b_Pusher$interconnect_Slide1_Black  :=  b_Pusher$Timer_Slide1_Black$Q ;
            END_IF
            IF  b_Pusher$interconnect_Slide1_Black  THEN
                 b_Pusher$_transit  := TRUE;
                 b_Pusher$_state  := Pusher_states_t#PusherY1_Move_Out_Black;
            END_IF

        Pusher_states_t#First_Slide_Timer_Metal:
             b_Pusher$_transit  := FALSE;
             b_Pusher$Timer_Slide1_Metal$IN  := TRUE;
             b_Pusher$Timer_Slide1_Metal$PT  :=  b_Pusher$Duration_Slide1_Metal ;
            IF  b_Pusher$Timer_Slide1_Metal$IN  THEN
                 b_Pusher$Timer_Slide1_Metal$Q  := ( b_Pusher$Timer_Slide1_Metal$ET  = USINT#0);
                IF ( b_Pusher$Timer_Slide1_Metal$ET  > USINT#0) THEN
                     b_Pusher$Timer_Slide1_Metal$ET  := ( b_Pusher$Timer_Slide1_Metal$ET  - USINT#1);
                ELSE
                     b_Pusher$Timer_Slide1_Metal$ET  := USINT#0;
                END_IF
            ELSE
                 b_Pusher$Timer_Slide1_Metal$Q  := FALSE;
                 b_Pusher$Timer_Slide1_Metal$ET  :=  b_Pusher$Timer_Slide1_Metal$PT ;
            END_IF
             b_Pusher$interconnect_Slide1_Metal  :=  b_Pusher$Timer_Slide1_Metal$Q ;
            IF  b_Pusher$interconnect_Slide1_Metal  THEN
                 b_Pusher$_transit  := TRUE;
                 b_Pusher$_state  := Pusher_states_t#PusherY1_Move_Out_Metal;
            END_IF

        Pusher_states_t#First_Slide_Timer_White:
             b_Pusher$_transit  := FALSE;
             b_Pusher$Timer_Slide1_White$IN  := TRUE;
             b_Pusher$Timer_Slide1_White$PT  :=  b_Pusher$Duration_Slide1_White ;
            IF  b_Pusher$Timer_Slide1_White$IN  THEN
                 b_Pusher$Timer_Slide1_White$Q  := ( b_Pusher$Timer_Slide1_White$ET  = USINT#0);
                IF ( b_Pusher$Timer_Slide1_White$ET  > USINT#0) THEN
                     b_Pusher$Timer_Slide1_White$ET  := ( b_Pusher$Timer_Slide1_White$ET  - USINT#1);
                ELSE
                     b_Pusher$Timer_Slide1_White$ET  := USINT#0;
                END_IF
            ELSE
                 b_Pusher$Timer_Slide1_White$Q  := FALSE;
                 b_Pusher$Timer_Slide1_White$ET  :=  b_Pusher$Timer_Slide1_White$PT ;
            END_IF
             b_Pusher$interconnect_Slide1_White  :=  b_Pusher$Timer_Slide1_White$Q ;
            IF  b_Pusher$interconnect_Slide1_White  THEN
                 b_Pusher$_transit  := TRUE;
                 b_Pusher$_state  := Pusher_states_t#PusherY1_Move_Out_White;
            END_IF

        Pusher_states_t#First_Slide_black_workpieces:
             b_Pusher$_transit  := FALSE;
            IF TRUE THEN
                 b_Pusher$_transit  := TRUE;
                 b_Pusher$_state  := Pusher_states_t#First_Slide_Timer_Black;
            END_IF

        Pusher_states_t#First_Slide_metal_workpieces:
             b_Pusher$_transit  := FALSE;
            IF TRUE THEN
                 b_Pusher$_transit  := TRUE;
                 b_Pusher$_state  := Pusher_states_t#First_Slide_Timer_Metal;
            END_IF

        Pusher_states_t#First_Slide_white_workpieces:
             b_Pusher$_transit  := FALSE;
            IF TRUE THEN
                 b_Pusher$_transit  := TRUE;
                 b_Pusher$_state  := Pusher_states_t#First_Slide_Timer_White;
            END_IF

        Pusher_states_t#Init:
             b_Pusher$_transit  := FALSE;
            IF  b_Pusher$StartVar  THEN
                 b_Pusher$_transit  := TRUE;
                 b_Pusher$_state  := Pusher_states_t#Interstep;
            END_IF

        Pusher_states_t#Interstep:
             b_Pusher$_transit  := FALSE;
             b_Pusher$PusherY1  := FALSE;
             b_Pusher$PusherY2  := FALSE;
             b_Pusher$interconnect2  := FALSE;
             b_Pusher$interconnect3  := FALSE;
             b_Pusher$StartVar  := FALSE;
             b_Pusher$interconnect_Slide1_Black  := FALSE;
             b_Pusher$interconnect_Slide2_Black  := FALSE;
             b_Pusher$interconnect_Slide1_White  := FALSE;
             b_Pusher$interconnect_Slide2_White  := FALSE;
             b_Pusher$interconnect_Slide1_Metal  := FALSE;
             b_Pusher$interconnect_Slide2_Metal  := FALSE;
            IF TRUE THEN
                 b_Pusher$_transit  := TRUE;
                 b_Pusher$_state  := Pusher_states_t#Interstep_2;
            END_IF

        Pusher_states_t#Interstep_2:
             b_Pusher$_transit  := FALSE;
            IF (( b_Pusher$SorterLightnessSensorPusher1  AND  b_Pusher$SorterCapacitiveSensorPusher1 ) AND ( b_Pusher$Priority_Var_Metal  > INT#0)) THEN
                 b_Pusher$_transit  := TRUE;
                 b_Pusher$_state  := Pusher_states_t#Check_For_Metal;
            ELSEIF ((NOT  b_Pusher$SorterLightnesssensorCraneInterfaceInverse  AND  b_Pusher$SorterLightbarrierCraneInterface ) AND ( b_Pusher$Priority_Var_Black  > INT#0)) THEN
                 b_Pusher$_transit  := TRUE;
                 b_Pusher$_state  := Pusher_states_t#Check_For_Black;
            ELSEIF (( b_Pusher$SorterLightnessSensorPusher1  AND NOT  b_Pusher$SorterCapacitiveSensorPusher1 ) AND ( b_Pusher$Priority_Var_White  > INT#0)) THEN
                 b_Pusher$_transit  := TRUE;
                 b_Pusher$_state  := Pusher_states_t#Check_For_White;
            END_IF

        Pusher_states_t#PusherY1_Move_In_Black:
             b_Pusher$_transit  := FALSE;
            IF (( b_Pusher$SorterPusher1MovedOut  = TRUE) AND ( b_Pusher$SorterPusher1MovedIn  = FALSE)) THEN
                 b_Pusher$PusherY1  := FALSE;
            END_IF
            IF  b_Pusher$SorterPusher1MovedIn  THEN
                 b_Pusher$_transit  := TRUE;
                 b_Pusher$_state  := Pusher_states_t#Reset_interconnect_Slide1_Black;
            END_IF

        Pusher_states_t#PusherY1_Move_In_Metal:
             b_Pusher$_transit  := FALSE;
            IF (( b_Pusher$SorterPusher1MovedOut  = TRUE) AND ( b_Pusher$SorterPusher1MovedIn  = FALSE)) THEN
                 b_Pusher$PusherY1  := FALSE;
            END_IF
            IF  b_Pusher$SorterPusher1MovedIn  THEN
                 b_Pusher$_transit  := TRUE;
                 b_Pusher$_state  := Pusher_states_t#Reset_interconnect_Slide1_Metal;
            END_IF

        Pusher_states_t#PusherY1_Move_In_White:
             b_Pusher$_transit  := FALSE;
            IF (( b_Pusher$SorterPusher1MovedOut  = TRUE) AND ( b_Pusher$SorterPusher1MovedIn  = FALSE)) THEN
                 b_Pusher$PusherY1  := FALSE;
            END_IF
            IF  b_Pusher$SorterPusher1MovedIn  THEN
                 b_Pusher$_transit  := TRUE;
                 b_Pusher$_state  := Pusher_states_t#Reset_interconnect_Slide1_White;
            END_IF

        Pusher_states_t#PusherY1_Move_Out_Black:
             b_Pusher$_transit  := FALSE;
            IF (( b_Pusher$SorterPusher1MovedOut  = FALSE) AND ( b_Pusher$SorterPusher1MovedIn  = TRUE)) THEN
                 b_Pusher$PusherY1  := TRUE;
            END_IF
            IF  b_Pusher$SorterPusher1MovedOut  THEN
                 b_Pusher$_transit  := TRUE;
                 b_Pusher$_state  := Pusher_states_t#Wait_Y1_Black;
            END_IF

        Pusher_states_t#PusherY1_Move_Out_Metal:
             b_Pusher$_transit  := FALSE;
            IF (( b_Pusher$SorterPusher1MovedOut  = FALSE) AND ( b_Pusher$SorterPusher1MovedIn  = TRUE)) THEN
                 b_Pusher$PusherY1  := TRUE;
            END_IF
            IF  b_Pusher$SorterPusher1MovedOut  THEN
                 b_Pusher$_transit  := TRUE;
                 b_Pusher$_state  := Pusher_states_t#Wait_Y1_Metal;
            END_IF

        Pusher_states_t#PusherY1_Move_Out_White:
             b_Pusher$_transit  := FALSE;
            IF (( b_Pusher$SorterPusher1MovedOut  = FALSE) AND ( b_Pusher$SorterPusher1MovedIn  = TRUE)) THEN
                 b_Pusher$PusherY1  := TRUE;
            END_IF
            IF  b_Pusher$SorterPusher1MovedOut  THEN
                 b_Pusher$_transit  := TRUE;
                 b_Pusher$_state  := Pusher_states_t#Wait_Y1_White;
            END_IF

        Pusher_states_t#PusherY2_Move_In_Black:
             b_Pusher$_transit  := FALSE;
            IF (( b_Pusher$SorterPusher2MovedOut  = TRUE) AND ( b_Pusher$SorterPusher2MovedIn  = FALSE)) THEN
                 b_Pusher$PusherY2  := FALSE;
            END_IF
            IF  b_Pusher$SorterPusher2MovedIn  THEN
                 b_Pusher$_transit  := TRUE;
                 b_Pusher$_state  := Pusher_states_t#Reset_interconnect_Slide2_Black;
            END_IF

        Pusher_states_t#PusherY2_Move_In_Metal:
             b_Pusher$_transit  := FALSE;
            IF (( b_Pusher$SorterPusher2MovedOut  = TRUE) AND ( b_Pusher$SorterPusher2MovedIn  = FALSE)) THEN
                 b_Pusher$PusherY2  := FALSE;
            END_IF
            IF  b_Pusher$SorterPusher2MovedIn  THEN
                 b_Pusher$_transit  := TRUE;
                 b_Pusher$_state  := Pusher_states_t#Reset_interconnect_Slide2_Metal;
            END_IF

        Pusher_states_t#PusherY2_Move_In_White:
             b_Pusher$_transit  := FALSE;
            IF (( b_Pusher$SorterPusher2MovedOut  = TRUE) AND ( b_Pusher$SorterPusher2MovedIn  = FALSE)) THEN
                 b_Pusher$PusherY2  := FALSE;
            END_IF
            IF  b_Pusher$SorterPusher2MovedIn  THEN
                 b_Pusher$_transit  := TRUE;
                 b_Pusher$_state  := Pusher_states_t#Reset_interconnect_Slide2_White;
            END_IF

        Pusher_states_t#PusherY2_Move_Out_Black:
             b_Pusher$_transit  := FALSE;
            IF (( b_Pusher$SorterPusher2MovedOut  = FALSE) AND ( b_Pusher$SorterPusher2MovedIn  = TRUE)) THEN
                 b_Pusher$PusherY2  := TRUE;
            END_IF
            IF  b_Pusher$SorterPusher2MovedOut  THEN
                 b_Pusher$_transit  := TRUE;
                 b_Pusher$_state  := Pusher_states_t#Wait_Y2_Black;
            END_IF

        Pusher_states_t#PusherY2_Move_Out_Metal:
             b_Pusher$_transit  := FALSE;
            IF (( b_Pusher$SorterPusher2MovedOut  = FALSE) AND ( b_Pusher$SorterPusher2MovedIn  = TRUE)) THEN
                 b_Pusher$PusherY2  := TRUE;
            END_IF
            IF  b_Pusher$SorterPusher2MovedOut  THEN
                 b_Pusher$_transit  := TRUE;
                 b_Pusher$_state  := Pusher_states_t#Wait_Y2_Metal;
            END_IF

        Pusher_states_t#PusherY2_Move_Out_White:
             b_Pusher$_transit  := FALSE;
            IF (( b_Pusher$SorterPusher2MovedOut  = FALSE) AND ( b_Pusher$SorterPusher2MovedIn  = TRUE)) THEN
                 b_Pusher$PusherY2  := TRUE;
            END_IF
            IF  b_Pusher$SorterPusher2MovedOut  THEN
                 b_Pusher$_transit  := TRUE;
                 b_Pusher$_state  := Pusher_states_t#Wait_Y2_White;
            END_IF

        Pusher_states_t#Reset_interconnect3:
             b_Pusher$_transit  := FALSE;
             b_Pusher$interconnect2  := FALSE;
             b_Pusher$Timer2$IN  := FALSE;
             b_Pusher$Timer2$PT  := USINT#0;
            IF  b_Pusher$Timer2$IN  THEN
                 b_Pusher$Timer2$Q  := ( b_Pusher$Timer2$ET  = USINT#0);
                IF ( b_Pusher$Timer2$ET  > USINT#0) THEN
                     b_Pusher$Timer2$ET  := ( b_Pusher$Timer2$ET  - USINT#1);
                ELSE
                     b_Pusher$Timer2$ET  := USINT#0;
                END_IF
            ELSE
                 b_Pusher$Timer2$Q  := FALSE;
                 b_Pusher$Timer2$ET  :=  b_Pusher$Timer2$PT ;
            END_IF
             b_Pusher$Slide3_black  := ( b_Pusher$Slide3_black  - INT#1);
             b_Pusher$Priority_Var_Black  := ( b_Pusher$Priority_Var_Black  - INT#1);
            IF TRUE THEN
                 b_Pusher$_transit  := TRUE;
                 b_Pusher$_state  := Pusher_states_t#Interstep_2;
            END_IF
